(* CODESYS project CommonTypesAndFunctions 1.1.0.5.library
   Description: Some things to collect...
      some based on OSCAT library.
      see www.oscat.de for here home
   Version: 1.1.0.5
   Title: Common Helper for development
   Author: Stefan Dreyer
   DocFormat: reStructuredText
   Placeholder: CommonTypesAndFunctions
   LanguageModelAttribute: qualified-access-only
   CompiledLibraryCompatibilityVersion: CODESYS V3.5 SP15 Patch 2
   Company: Stefan Dreyer
   DefaultNamespace: CommonTypesAndFunctions

Project tree, tasks and I/O mapping:
  libraries: CAA Types Extern, * (CAA Technical Workgroup); CAA Behaviour Model, * (CAA Technical Workgroup); CAA FB Factory, * (CAA Technical Workgroup); SysTypes Interfaces, 3.5.2.0 (System); Time and Date, 3.5.7.0 (3S - Smart Software Solutions GmbH); SysTarget, 3.5.5.0 (System); SysMem, 3.5.12.0 (System); Standard, 3.5.15.0 (System); CmpErrors2 Interfaces, 3.5.15.0 (System); SysSem, 3.5.16.0 (System); SysProcess, 3.5.16.0 (System); Standard64, 3.5.16.0 (System); SysSocket2, 3.5.16.10 (System); CmpX509Cert, 3.5.15.0 (System); CmpTls, 3.5.15.0 (System); Base Interfaces, 3.5.2.0 (System); SysSocket, 3.5.15.0 (System); OSCAT Basic Extensions, 1.0.0.0 (Stefan Dreyer); BASIC, 3.3.4.0 (OSCAT); BUILDING, 1.0.0.1 (OSCAT); OSCAT Network Types, 1.0.0.1 (Stefan Dreyer)
  Common/
    Enums/
      data type ERROR
      data type VAR_TYPES
    Function Blocks/
      function block IP_CONTROL [ST]
      function block TIME_DATE_IMPULS [ST]
      function block TestString [ST]
      function block IP_CONTROL_TLS [ST]
      function block CounterToActuall [ST]: CounterInit, SetCounterResetImp
      function block StringImpact [ST]
      function block GetInstanceName [ST]: GetInstanceTopic, ReduceToLastNLevels, getLastName, GetName
      function block RELAIS_OUT_16_TRANSLATOR [ST]
      function block SmartDim [ST]
      function block Spratzel [ST]: setRand
      function block Rand [ST]: getRand
      Tests/
        function block TestNames1 [ST]
        function block TestInstanceName [ST]: FB_Init
        function block TestAnyX [ST]
      function block UpDown [ST]
      function block BLIND_INPUT_PERS [ST]
      function block BLIND_CONTROL_S_PERS [ST]
      function block BLIND_INPUT_EXT_PERS [ST]
      function block DivideByN [ST]
    Functions/
      function GET_DNS_IP [ST]
      function GetChar [ST]
      function find [ST]
      function len [ST]
      function concat [ST]
      function ResolveIPAddr [ST]
      function CheckDeltaValue [ST]
      function GetValueFromPointer [ST]
      function GetValueString [ST]
      function test [ST]
      function StrEquals [ST]
      function StrEqualsAtStart [ST]
      function GetValueFromStringPt [ST]
      function StrEqualsAtStartWithDelimiter [ST]
      function FindLastDot [ST]
      function MakeAllTypesPointer [ST]
      function GetJSONValue [ST]
      function Steps [ST]
      function GetValueStringFaktor [ST]
      function unionAdd [ST]
      function unionSub [ST]
      function unionMul [ST]
      function unionDiv [ST]
      function unionLimit [ST]
      function uint_to_Union [ST]
      function ScaleAllTypesUnion [ST]
      function AnyToUnion [ST]
      function unionToAny [ST]
      function checkJSON [ST]
    GlobalConstants/
      global variables MyConstants
    GlobalVariables/
      global variables Variables
    Interfaces/
    Structs/
      data type SMART_DIMM
      data type SMART_DIMM_ELEMENT
      data type IP_C_EXT
    Templates/
      Behaviour Model/
        function block ETrigA_Temp [ST]: prvAbort, prvCyclicAction, prvResetOutputs, prvStart
        function block ETrigTlA_Temp [ST]: prvAbort, prvCyclicAction, prvResetOutputs, prvStart
        function block ETrigTl_Temp [ST]: prvAbort, prvCyclicAction, prvResetOutputs, prvStart
        function block ETrigToA_Temp [ST]: prvAbort, prvCyclicAction, prvResetOutputs, prvStart
        function block ETrigToTlA_Temp [ST]: prvAbort, prvCyclicAction, prvResetOutputs, prvStart
        function block ETrigToTl_Temp [ST]: prvAbort, prvCyclicAction, prvResetOutputs, prvStart
        function block ETrigTo_Temp [ST]: prvAbort, prvCyclicAction, prvResetOutputs, prvStart
        function block ETrig_Temp [ST]: prvAbort, prvCyclicAction, prvResetOutputs, prvStart
        function block LTrig_Temp [ST]: prvAbort, prvCyclicAction, prvResetOutputs, prvStart
      FB Factory/
        function block CustomData [ST]
        function block CustomFB [ST]: prvInstInit
        function block CustomFBFactory_heap [ST]: Create, prvInstCount, prvInstPoolExtendsFactor, prvInstSize
        function block CustomFBFactory_static [ST]: Create, prvInstPoolAdr, prvInstPoolSize, prvInstSize
    Types/
      data type ALL_TYPES_UNION
      data type ALL_TYPES_UNION_POINTER
      data type EEPROM_DATA
      data type TIME_DATE_IMPULS_DATA
      data type TLS_CONFIG
      data type PWConfigs
      data type ENVIRONMENT_DATA
*)

// Common/Enums/ERROR
{attribute 'qualified_only'}
//{attribute 'conditionalshow'}
//{attribute 'conditionalshow' := 'SomeText'}
//{attribute 'hide'}
TYPE ERROR : (NO_ERROR, TIME_OUT); END_TYPE

// Common/Types/ALL_TYPES_UNION
TYPE ALL_TYPES_UNION :
UNION
	SINT_T:SINT;
	USINT_T:USINT;
	INT_T:INT;
	UINT_T:UINT;
	LINT_T:LINT;
	ULINT_T:ULINT;
	DINT_T:DINT;
	UDINT_T:UDINT;
	REAL_T:REAL;
	LREAL_T:LREAL;
	BYTE_T:BYTE;
	WORD_T:WORD;
	DWORD_T:DWORD;
	LWORD_T:LWORD;
	DT_T:DT;
	TIME_T:TIME;
	LTIME_T:LTIME;
	TOD_T:TOD;
	TOD_T2:ARRAY[0..1]OF TOD;
	DATE_T:DATE;
	BYTE_ARRAY:ARRAY[0..7]OF BYTE;
	BOOL_T:BOOL;
	
	//don't use strings UNION would be TO big....
END_UNION
END_TYPE

// Common/Types/ALL_TYPES_UNION_POINTER
TYPE ALL_TYPES_UNION_POINTER :
UNION
	POINTER_TO_SINT_T:POINTER TO SINT;
	POINTER_TO_USINT_T:POINTER TO USINT;
	POINTER_TO_INT_T:POINTER TO INT;
	POINTER_TO_UINT_T:POINTER TO UINT;
	POINTER_TO_LINT_T:POINTER TO LINT;
	POINTER_TO_ULINT_T:POINTER TO ULINT;
	POINTER_TO_DINT_T:POINTER TO DINT;
	POINTER_TO_UDINT_T:POINTER TO UDINT;
	POINTER_TO_REAL_T:POINTER TO REAL;
	POINTER_TO_LREAL_T:POINTER TO LREAL;
	POINTER_TO_BYTE_T:POINTER TO BYTE;
	POINTER_TO_WORD_T:POINTER TO WORD;
	POINTER_TO_DWORD_T:POINTER TO DWORD;
	POINTER_TO_LWORD_T:POINTER TO LWORD;
	POINTER_TO_DT_T:POINTER TO DT;
	POINTER_TO_TIME_T:POINTER TO TIME;
	POINTER_TO_LTIME_T:POINTER TO LTIME;
	POINTER_TO_TOD_T:POINTER TO TOD;
	POINTER_TO_TOD_T2:POINTER TO ARRAY[0..1]OF TOD;
	POINTER_TO_DATE_T:POINTER TO DATE;
	POINTER_TO_BYTE_ARRAY_T:POINTER TO ARRAY[0..7]OF BYTE;
	POINTER_TO_BOOL_T:POINTER TO BOOL;
	POINTER_TO_STRING_T: POINTER TO STRING(2000);

END_UNION
END_TYPE

// Common/Types/EEPROM_DATA
TYPE EEPROM_DATA :
STRUCT
	//FB_NO_AUTO:UINT;//auto createt FB NO, not possible because of multitasking ... so bad...
	FB_NO_IN:UINT;//allways check FB_IN_NO to be 0!!! so the EEPROM is free to do something!
	FB_NO_OUT:UINT;
	PAGE_IN:ARRAY[0..128-1] OF BYTE;
	PAGE_OUT:ARRAY[0..128-1] OF BYTE;
	READ_PAGE: BOOL;
	WRITE_PAGE: BOOL;
	ADDRESS_PAGE: UINT;
	ADDRESS_VALUE: UINT;
	VALUE_IN:ALL_TYPES_UNION;
	VALUE_OUT:ALL_TYPES_UNION; 
	READ_VALUE: BOOL;
	WRITE_VALUE: BOOL;
	PAGE_SIZE:UINT:=128;
	SIZE_OF_VALUE:UINT;
	SEMAPHORE:SysSem.RTS_IEC_HANDLE; //Semaphore for Consistence for EEPROM DATA is bus is out of main task
	HANDLE_VALID: BOOL;

END_STRUCT
END_TYPE

// Common/Types/TIME_DATE_IMPULS_DATA
TYPE TIME_DATE_IMPULS_DATA :
STRUCT
	
	IMP:BOOL;//1s impulse
	UDT:DT;//World Time
	SYSTEM_TIME:DT;//Time on SYSTEM
	TIME_IO:BOOL;//TIME IS I.O.
	TD_TIME:OSCAT_BASIC.SDT;
	//impulse at 00:00:00
	DAY_CHANGE:BOOL;
END_STRUCT
END_TYPE

// Common/Types/TLS_CONFIG
TYPE TLS_CONFIG :
STRUCT
	//see CmpTls for Doku of Method, initialisied to work as client
	tlsMethod: CmpTls.CmpTlsMethod := CmpTls.CmpTlsMethod.TLSv2_CLIENT;
	//List of allowed ciphers, initialised to medium, see openSSL for cipherList config
	chiperList:STRING(255) := 'HIGH';
	//certificates and ca still not supportet by CmpTls. So initialised to dont use certificats....
	{info 'here to implement certificate use'}
	verifyMode:DWORD := CmpTls.CmpTlsConstants.TLS_VERIFY_CLIENT_ONCE;
	
END_STRUCT
END_TYPE

// Common/Enums/VAR_TYPES
{attribute 'qualified_only'}
{attribute 'strict'}
TYPE VAR_TYPES :
(
	//enum_member := 0
	SINT_T, USINT_T, INT_T, UINT_T, DINT_T, UDINT_T, 
				LINT_T, ULINT_T, REAL_T, LREAL_T, BYTE_T, WORD_T,
				DWORD_T, LWORD_T, DT_T, TIME_T, TOD_T, TOD2_T, DATE_T, ARRAY_T, BOOL_T,
				STRING_T, LTIME_T
);
END_TYPE

// Common/Types/PWConfigs
TYPE PWConfigs :
STRUCT
PointerTo:ALL_TYPES_UNION_POINTER;
//PointerTo1:POINTER TO BYTE;
ValueType:VAR_TYPES;
NeedsMQTT:BOOL;
NeedsDB:BOOL;
MQTTTopic:POINTER TO STRING;
MQTTName:POINTER TO STRING;
MQTTDiff:UINT;
MQTTDezimal:INT;
MQTTTime:TIME;
MQTTRetain:BOOL;
MQTTQoS:SD_MQTT.QoS;
DBName:STRING;
DBNum:UINT;




END_STRUCT
END_TYPE

// Common/Structs/SMART_DIMM
TYPE SMART_DIMM :
STRUCT
	values:ARRAY[0..MyConstants.SMART_DIMM_STAGES-1] OF SMART_DIMM_ELEMENT;
END_STRUCT
END_TYPE

// Common/Structs/SMART_DIMM_ELEMENT
TYPE SMART_DIMM_ELEMENT :
STRUCT
	RunTime:TIME;//duration off effect
	DeltaOut:UINT;//Delta for Output
	_from:LREAL;
	_to:LREAL;
	Value:UINT;
END_STRUCT
END_TYPE

// Common/Types/ENVIRONMENT_DATA
TYPE ENVIRONMENT_DATA :
STRUCT
	//Possible Data from BME280 from Bosch Sensor Tec
	//using -->LREAL;
	Temperatur:LREAL;//using -->LREAL;
	//using -->LREAL;
	Humidity:LREAL;//using -->LREAL;
	//using -->LREAL;
	Pressure: LREAL;//using -->LREAL;
	//using -->REAL;
	absHumidity:REAL;//using -->REAL;
	//using -->REAL;
	dewPoint:REAL;//using -->REAL;


END_STRUCT
END_TYPE

// Common/Structs/IP_C_EXT
TYPE IP_C_EXT EXTENDS OSCAT_NETWORK_TYPES.IP_C :
STRUCT
	ResultSend:SysTypes.RTS_IEC_RESULT; 			(*Result of TCP Send call*)
	ResultReceive:SysTypes.RTS_IEC_RESULT;		(*Result of TCP Receive call*)
END_STRUCT
END_TYPE

// Common/GlobalConstants/MyConstants
{attribute 'qualified_only'}
//{attribute 'conditionalshow'}
//{attribute 'conditionalshow' := 'SomeText'}
//{attribute 'hide'}
VAR_GLOBAL CONSTANT
	gc_iDummy : INT := 42; /// This is a dummy global constant variable
	//Countrs in coutr ;)
	COUNTER_COUNT:UINT:=5;
	SMART_DIMM_STAGES:UINT:=5;
END_VAR

// Common/GlobalVariables/Variables
{attribute 'qualified_only'}
//{attribute 'conditionalshow'}
//{attribute 'conditionalshow' := 'SomeText'}
//{attribute 'hide'}
VAR_GLOBAL
	g_iDummy : INT; /// This is a dummy global variable
END_VAR

// Common/Templates/Behaviour Model/ETrigA_Temp
//{attribute 'hide_all_locals'}
//{attribute 'conditionalshow_all_locals' := 'SomeText'}
//{attribute 'conditionalshow_all_locals'}
//{attribute 'conditionalshow' := 'SomeText'}
//{attribute 'conditionalshow'}
//{attribute 'hide'}
FUNCTION_BLOCK ETrigA_Temp EXTENDS CBM.ETrigA
VAR_INPUT
	(* specific Inputs *)
END_VAR
VAR_OUTPUT
	eError : ERROR;
	(* specific Outputs *)
END_VAR
VAR
	(* specific vars *)
END_VAR

SUPER^();
IF iError = CBM.ERROR.TIME_OUT THEN
	eError := ERROR.TIME_OUT;
ELSE
	eError := iError;
END_IF

{attribute 'hide'}
METHOD prvAbort : BOOL
VAR_INPUT
END_VAR
VAR
END_VAR
IF xError THEN (* abort because of error *)
	(* TODO: insert specific Code here *)
ELSE (* user abort *)
	(* TODO: insert specific Code here *)
END_IF
xAbortInProgress:= FALSE;
END_METHOD

{attribute 'hide'}
METHOD prvCyclicAction : BOOL
VAR_INPUT
END_VAR
VAR
END_VAR
(* TODO: insert specific Code here *)
xDone:= TRUE;
(* if an error occurs, set iError to a value else than zero instead of xDone:= TRUE *)
(* to keep repeat loop *)
END_METHOD

{attribute 'hide'}
METHOD prvResetOutputs : BOOL
VAR_INPUT
END_VAR
VAR
END_VAR
(* TODO: insert specific Code here *)
SUPER^.prvResetOutputs();
END_METHOD

{attribute 'hide'}
METHOD prvStart : BOOL
VAR_INPUT
END_VAR
VAR
END_VAR
(* this code is called, when the application is started (rising edge of xExecute *)
(* TODO: copy specific input variables into local copies *)
(* TODO: insert specific Code here *)
;
END_METHOD

END_FUNCTION_BLOCK

// Common/Templates/Behaviour Model/ETrigTlA_Temp
//{attribute 'hide_all_locals'}
//{attribute 'conditionalshow_all_locals' := 'SomeText'}
//{attribute 'conditionalshow_all_locals'}
//{attribute 'conditionalshow' := 'SomeText'}
//{attribute 'conditionalshow'}
//{attribute 'hide'}
FUNCTION_BLOCK ETrigTlA_Temp EXTENDS CBM.ETrigTlA
VAR_INPUT
	(* specific Inputs *)
END_VAR
VAR_OUTPUT
	eError : ERROR;
	(* specific Outputs *)
END_VAR
VAR
	(* specific vars *)
END_VAR

SUPER^();
IF iError = CBM.ERROR.TIME_OUT THEN
	eError := ERROR.TIME_OUT;
ELSE
	eError := iError;
END_IF

{attribute 'hide'}
METHOD prvAbort : BOOL
VAR_INPUT
END_VAR
VAR
END_VAR
IF xError THEN (* abort because of error *)
	(* TODO: insert specific Code here *)
ELSE (* user abort *)
	(* TODO: insert specific Code here *)
END_IF
xAbortInProgress:= FALSE;
END_METHOD

{attribute 'hide'}
METHOD prvCyclicAction : BOOL
VAR_INPUT
END_VAR
VAR
END_VAR
(* TODO: insert specific Code here *)
xDone:= TRUE;
(* if an error occurs, set iError to a value else than zero instead of xDone:= TRUE *)
(* to keep repeat loop *)
END_METHOD

{attribute 'hide'}
METHOD prvResetOutputs : BOOL
VAR_INPUT
END_VAR
VAR
END_VAR
(* TODO: insert specific Code here *)
SUPER^.prvResetOutputs();
END_METHOD

{attribute 'hide'}
METHOD prvStart : BOOL
VAR_INPUT
END_VAR
VAR
END_VAR
(* this code is called, when the application is started (rising edge of xExecute *)
(* TODO: copy specific input variables into local copies *)
(* TODO: insert specific Code here *)
;
END_METHOD

END_FUNCTION_BLOCK

// Common/Templates/Behaviour Model/ETrigTl_Temp
//{attribute 'hide_all_locals'}
//{attribute 'conditionalshow_all_locals' := 'SomeText'}
//{attribute 'conditionalshow_all_locals'}
//{attribute 'conditionalshow' := 'SomeText'}
//{attribute 'conditionalshow'}
//{attribute 'hide'}
FUNCTION_BLOCK ETrigA_Temp EXTENDS CBM.ETrigTl
VAR_INPUT
	(* specific Inputs *)
END_VAR
VAR_OUTPUT
	eError : ERROR;
	(* specific Outputs *)
END_VAR
VAR
	(* specific vars *)
END_VAR

SUPER^();
IF iError = CBM.ERROR.TIME_OUT THEN
	eError := ERROR.TIME_OUT;
ELSE
	eError := iError;
END_IF

{attribute 'hide'}
METHOD prvAbort : BOOL
VAR_INPUT
END_VAR
VAR
END_VAR
IF xError THEN (* abort because of error *)
	(* TODO: insert specific Code here *)
ELSE (* user abort *)
	(* TODO: insert specific Code here *)
END_IF
xAbortInProgress:= FALSE;
END_METHOD

{attribute 'hide'}
METHOD prvCyclicAction : BOOL
VAR_INPUT
END_VAR
VAR
END_VAR
(* TODO: insert specific Code here *)
xDone:= TRUE;
(* if an error occurs, set iError to a value else than zero instead of xDone:= TRUE *)
(* to keep repeat loop *)
END_METHOD

{attribute 'hide'}
METHOD prvResetOutputs : BOOL
VAR_INPUT
END_VAR
VAR
END_VAR
(* TODO: insert specific Code here *)
SUPER^.prvResetOutputs();
END_METHOD

{attribute 'hide'}
METHOD prvStart : BOOL
VAR_INPUT
END_VAR
VAR
END_VAR
(* this code is called, when the application is started (rising edge of xExecute *)
(* TODO: copy specific input variables into local copies *)
(* TODO: insert specific Code here *)
;
END_METHOD

END_FUNCTION_BLOCK

// Common/Templates/Behaviour Model/ETrigToA_Temp
//{attribute 'hide_all_locals'}
//{attribute 'conditionalshow_all_locals' := 'SomeText'}
//{attribute 'conditionalshow_all_locals'}
//{attribute 'conditionalshow' := 'SomeText'}
//{attribute 'conditionalshow'}
//{attribute 'hide'}
FUNCTION_BLOCK ETrigToA_Temp EXTENDS CBM.ETrigToA
VAR_INPUT
	(* specific Inputs *)
END_VAR
VAR_OUTPUT
	eError : ERROR;
	(* specific Outputs *)
END_VAR
VAR
	(* specific vars *)
END_VAR

SUPER^();
IF iError = CBM.ERROR.TIME_OUT THEN
	eError := ERROR.TIME_OUT;
ELSE
	eError := iError;
END_IF

{attribute 'hide'}
METHOD prvAbort : BOOL
VAR_INPUT
END_VAR
VAR
END_VAR
IF xError THEN (* abort because of error *)
	(* TODO: insert specific Code here *)
ELSE (* user abort *)
	(* TODO: insert specific Code here *)
END_IF
xAbortInProgress:= FALSE;
END_METHOD

{attribute 'hide'}
METHOD prvCyclicAction : BOOL
VAR_INPUT
END_VAR
VAR
END_VAR
(* TODO: insert specific Code here *)
xDone:= TRUE;
(* if an error occurs, set iError to a value else than zero instead of xDone:= TRUE *)
END_METHOD

{attribute 'hide'}
METHOD prvResetOutputs : BOOL
VAR_INPUT
END_VAR
VAR
END_VAR
(* TODO: insert specific Code here *)
SUPER^.prvResetOutputs();
END_METHOD

{attribute 'hide'}
METHOD prvStart : BOOL
VAR_INPUT
END_VAR
VAR
END_VAR
(* this code is called, when the application is started (rising edge of xExecute *)
(* TODO: copy specific input variables into local copies *)
(* TODO: insert specific Code here *)
;
END_METHOD

END_FUNCTION_BLOCK

// Common/Templates/Behaviour Model/ETrigToTlA_Temp
//{attribute 'hide_all_locals'}
//{attribute 'conditionalshow_all_locals' := 'SomeText'}
//{attribute 'conditionalshow_all_locals'}
//{attribute 'conditionalshow' := 'SomeText'}
//{attribute 'conditionalshow'}
//{attribute 'hide'}
FUNCTION_BLOCK ETrigToTlA_Temp EXTENDS CBM.ETrigToTlA
VAR_INPUT
	(* specific Inputs *)
END_VAR
VAR_OUTPUT
	eError : ERROR;
	(* specific Outputs *)
END_VAR
VAR
	(* specific vars *)
END_VAR

SUPER^();
IF iError = CBM.ERROR.TIME_OUT THEN
	eError := ERROR.TIME_OUT;
ELSE
	eError := iError;
END_IF

{attribute 'hide'}
METHOD prvAbort : BOOL
VAR_INPUT
END_VAR
VAR
END_VAR
IF xError THEN (* abort because of error *)
	(* TODO: insert specific Code here *)
ELSE (* user abort *)
	(* TODO: insert specific Code here *)
END_IF
xAbortInProgress:= FALSE;
END_METHOD

{attribute 'hide'}
METHOD prvCyclicAction : BOOL
VAR_INPUT
END_VAR
VAR
END_VAR
(* TODO: insert specific Code here *)
xDone:= TRUE;
(* if an error occurs, set iError to a value else than zero instead of xDone:= TRUE *)
(* to keep repeat loop *)
END_METHOD

{attribute 'hide'}
METHOD prvResetOutputs : BOOL
VAR_INPUT
END_VAR
VAR
END_VAR
(* TODO: insert specific Code here *)
SUPER^.prvResetOutputs();
END_METHOD

{attribute 'hide'}
METHOD prvStart : BOOL
VAR_INPUT
END_VAR
VAR
END_VAR
(* this code is called, when the application is started (rising edge of xExecute *)
(* TODO: copy specific input variables into local copies *)
(* TODO: insert specific Code here *)
;
END_METHOD

END_FUNCTION_BLOCK

// Common/Templates/Behaviour Model/ETrigToTl_Temp
//{attribute 'hide_all_locals'}
//{attribute 'conditionalshow_all_locals' := 'SomeText'}
//{attribute 'conditionalshow_all_locals'}
//{attribute 'conditionalshow' := 'SomeText'}
//{attribute 'conditionalshow'}
//{attribute 'hide'}
FUNCTION_BLOCK ETrigToTl_Temp EXTENDS CBM.ETrigToTl
VAR_INPUT
	(* specific Inputs *)
END_VAR
VAR_OUTPUT
	eError : ERROR;
	(* specific Outputs *)
END_VAR
VAR
	(* specific vars *)
END_VAR

SUPER^();
IF iError = CBM.ERROR.TIME_OUT THEN
	eError := ERROR.TIME_OUT;
ELSE
	eError := iError;
END_IF

{attribute 'hide'}
METHOD prvAbort : BOOL
VAR_INPUT
END_VAR
VAR
END_VAR
IF xError THEN (* abort because of error *)
	(* TODO: insert specific Code here *)
ELSE (* user abort *)
	(* TODO: insert specific Code here *)
END_IF
xAbortInProgress:= FALSE;
END_METHOD

{attribute 'hide'}
METHOD prvCyclicAction : BOOL
VAR_INPUT
END_VAR
VAR
END_VAR
(* TODO: insert specific Code here *)
xDone:= TRUE;
(* if an error occurs, set iError to a value else than zero instead of xDone:= TRUE *)
(* to keep repeat loop *)
END_METHOD

{attribute 'hide'}
METHOD prvResetOutputs : BOOL
VAR_INPUT
END_VAR
VAR
END_VAR
(* TODO: insert specific Code here *)
SUPER^.prvResetOutputs();
END_METHOD

{attribute 'hide'}
METHOD prvStart : BOOL
VAR_INPUT
END_VAR
VAR
END_VAR
(* this code is called, when the application is started (rising edge of xExecute *)
(* TODO: copy specific input variables into local copies *)
(* TODO: insert specific Code here *)
;
END_METHOD

END_FUNCTION_BLOCK

// Common/Templates/Behaviour Model/ETrigTo_Temp
//{attribute 'hide_all_locals'}
//{attribute 'conditionalshow_all_locals' := 'SomeText'}
//{attribute 'conditionalshow_all_locals'}
//{attribute 'conditionalshow' := 'SomeText'}
//{attribute 'conditionalshow'}
//{attribute 'hide'}
FUNCTION_BLOCK ETrigTo_Temp EXTENDS CBM.ETrigTo
VAR_INPUT
	(* specific Inputs *)
END_VAR
VAR_OUTPUT
	eError : ERROR;
	(* specific Outputs *)
END_VAR
VAR
	(* specific vars *)
END_VAR

SUPER^();
IF iError = CBM.ERROR.TIME_OUT THEN
	eError := ERROR.TIME_OUT;
ELSE
	eError := iError;
END_IF

{attribute 'hide'}
METHOD prvAbort : BOOL
VAR_INPUT
END_VAR
VAR
END_VAR
IF xError THEN (* abort because of error *)
	(* TODO: insert specific Code here *)
ELSE (* user abort *)
	(* TODO: insert specific Code here *)
END_IF
xAbortInProgress:= FALSE;
END_METHOD

{attribute 'hide'}
METHOD prvCyclicAction : BOOL
VAR_INPUT
END_VAR
VAR
END_VAR
(* TODO: insert specific Code here *)
xDone:= TRUE;
(* if an error occurs, set iError to a value else than zero instead of xDone:= TRUE *)
(* to keep repeat loop *)
END_METHOD

{attribute 'hide'}
METHOD prvResetOutputs : BOOL
VAR_INPUT
END_VAR
VAR
END_VAR
(* TODO: insert specific Code here *)
SUPER^.prvResetOutputs();
END_METHOD

{attribute 'hide'}
METHOD prvStart : BOOL
VAR_INPUT
END_VAR
VAR
END_VAR
(* this code is called, when the application is started (rising edge of xExecute *)
(* TODO: copy specific input variables into local copies *)
(* TODO: insert specific Code here *)
;
END_METHOD

END_FUNCTION_BLOCK

// Common/Templates/Behaviour Model/ETrig_Temp
//{attribute 'hide_all_locals'}
//{attribute 'conditionalshow_all_locals' := 'SomeText'}
//{attribute 'conditionalshow_all_locals'}
//{attribute 'conditionalshow' := 'SomeText'}
//{attribute 'conditionalshow'}
//{attribute 'hide'}
FUNCTION_BLOCK ETrig_Temp EXTENDS CBM.ETrig
VAR_INPUT
	(* specific Inputs *)
END_VAR
VAR_OUTPUT
	eError : ERROR;
	(* specific Outputs *)
END_VAR
VAR
	(* specific vars *)
END_VAR

SUPER^();
IF iError = CBM.ERROR.TIME_OUT THEN
	eError := ERROR.TIME_OUT;
ELSE
	eError := iError;
END_IF

{attribute 'hide'}
METHOD prvAbort : BOOL
VAR_INPUT
END_VAR
VAR
END_VAR
IF xError THEN (* abort because of error *)
	(* TODO: insert specific Code here *)
ELSE (* user abort *)
	(* TODO: insert specific Code here *)
END_IF
xAbortInProgress:= FALSE;
END_METHOD

{attribute 'hide'}
METHOD prvCyclicAction : BOOL
VAR_INPUT
END_VAR
VAR
END_VAR
(* TODO: insert specific Code here *)
xDone:= TRUE;
(* if an error occurs, set iError to a value else than zero instead of xDone:= TRUE *)
(* to keep repeat loop *)
END_METHOD

{attribute 'hide'}
METHOD prvResetOutputs : BOOL
VAR_INPUT
END_VAR
VAR
END_VAR
(* TODO: insert specific Code here *)
SUPER^.prvResetOutputs();
END_METHOD

{attribute 'hide'}
METHOD prvStart : BOOL
VAR_INPUT
END_VAR
VAR
END_VAR
(* this code is called, when the application is started (rising edge of xExecute *)
(* TODO: copy specific input variables into local copies *)
(* TODO: insert specific Code here *)
;
END_METHOD

END_FUNCTION_BLOCK

// Common/Templates/Behaviour Model/LTrig_Temp
//{attribute 'hide_all_locals'}
//{attribute 'conditionalshow_all_locals' := 'SomeText'}
//{attribute 'conditionalshow_all_locals'}
//{attribute 'conditionalshow' := 'SomeText'}
//{attribute 'conditionalshow'}
//{attribute 'hide'}
FUNCTION_BLOCK LTrig_Temp EXTENDS CBM.LTrig
VAR_INPUT
	(* specific Inputs *)
END_VAR
VAR_OUTPUT
	eError : ERROR;
	(* specific Outputs *)
END_VAR
VAR
	(* specific vars *)
END_VAR

SUPER^();
IF iError = CBM.ERROR.TIME_OUT THEN
	eError := ERROR.TIME_OUT;
ELSE
	eError := iError;
END_IF

{attribute 'hide'}
METHOD prvAbort : BOOL
VAR_INPUT
END_VAR
VAR
END_VAR
IF xError THEN (* abort because of error *)
	(* TODO: insert specific Code here *)
ELSE (* user abort *)
	(* TODO: insert specific Code here *)
END_IF
xAbortInProgress:= FALSE;
END_METHOD

{attribute 'hide'}
METHOD prvCyclicAction : BOOL
VAR_INPUT
END_VAR
VAR
END_VAR
(* TODO: insert specific Code here *)
xDone:= TRUE;
(* if an error occurs, set iError to a value else than zero instead of xDone:= TRUE *)
(* to keep repeat loop *)
END_METHOD

{attribute 'hide'}
METHOD prvResetOutputs : BOOL
VAR_INPUT
END_VAR
VAR
END_VAR
(* TODO: insert specific Code here *)
SUPER^.prvResetOutputs();
END_METHOD

{attribute 'hide'}
METHOD prvStart : BOOL
VAR_INPUT
END_VAR
VAR
END_VAR
(* this code is called, when the application is started (rising edge of xExecute *)
(* TODO: copy specific input variables into local copies *)
(* TODO: insert specific Code here *)
;
END_METHOD

END_FUNCTION_BLOCK

// Common/Templates/FB Factory/CustomData
// This is a container to carry init data from the Create methode of the factory
// to the prvInstInit methode of the new generated function block instance
{attribute 'enable_dynamic_creation'}
//{attribute 'hide_all_locals'}
//{attribute 'conditionalshow_all_locals' := 'SomeText'}
//{attribute 'conditionalshow_all_locals'}
//{attribute 'conditionalshow' := 'SomeText'}
//{attribute 'conditionalshow'}
//{attribute 'hide'}
FUNCTION_BLOCK CustomData EXTENDS FBF.InstanceData
VAR_INPUT
	(* Todo: Add your application specific data as input variables *)
END_VAR

(* !! Do not add any executable code here !! *)
SUPER^();

END_FUNCTION_BLOCK

// Common/Templates/FB Factory/CustomFB
{attribute 'enable_dynamic_creation'}
//{attribute 'hide_all_locals'}
//{attribute 'conditionalshow_all_locals' := 'SomeText'}
//{attribute 'conditionalshow_all_locals'}
//{attribute 'conditionalshow' := 'SomeText'}
//{attribute 'conditionalshow'}
//{attribute 'hide'}
FUNCTION_BLOCK CustomFB EXTENDS FBF.InstanceBase;
VAR_INPUT
END_VAR
VAR_OUTPUT
END_VAR
VAR
END_VAR

SUPER^();

// This methode is called from the factory to give a chance
// to initialize the new fb instance with the content of itfData
//{attribute 'hide_all_locals'}
//{attribute 'conditionalshow_all_locals' := 'SomeText'}
//{attribute 'conditionalshow_all_locals'}
//{attribute 'conditionalshow' := 'SomeText'}
//{attribute 'conditionalshow'}
//{attribute 'hide'}
METHOD prvInstInit : FBF.ERROR
VAR_INPUT
	itfData : FBF.IData; 
END_VAR
VAR
	pData : POINTER TO CustomData;
	xOk : BOOL;
END_VAR
SUPER^.prvInstInit(itfData);
xOk := __QUERYPOINTER(itfData, pData);
IF xOk THEN
	(* THIS^.iLocalVar := pData^.iInitValue *);
END_IF
END_METHOD

END_FUNCTION_BLOCK

// Common/Templates/FB Factory/CustomFBFactory_heap
// This is a template for a factory with an heap based extendable memory pool
{attribute 'enable_dynamic_creation'}
//{attribute 'hide_all_locals'}
//{attribute 'conditionalshow_all_locals' := 'SomeText'}
//{attribute 'conditionalshow_all_locals'}
//{attribute 'conditionalshow' := 'SomeText'}
//{attribute 'conditionalshow'}
//{attribute 'hide'}
FUNCTION_BLOCK CustomFBFactory_heap EXTENDS FBF.FactoryBase
VAR
END_VAR

SUPER^();

(* Please replace CustonFB with your specific function block type *)
(* There is no need to change anything else !!! *)
METHOD Create : POINTER TO CustomFB
VAR_INPUT
	itfData : FBF.IData;
END_VAR
VAR_OUTPUT
	eError : FBF.ERROR;
END_VAR
VAR
	hInst : CAA.HANDLE;
	itfInst : FBF.IInstance;
	xOk : BOOL;
END_VAR
(* !!! This code must not be subject to change !!! *)
hInst := SUPER^.prvAllocInstMem(eError => eError);
Create := SUPER^.prvGetInstPointer(hInst);
IF Create <> 0 AND eError = FBF.ERROR.NO_ERROR THEN

	{implicit on}
	Create^.__vfInit();
	Create^.FB_Init(TRUE, FALSE);
	{implicit off}

	xOk := __QUERYINTERFACE(Create^, itfInst);
	IF xOk THEN
		xOk := SUPER^.prvInstInit(itfInst, hInst, itfData, eError=>eError);
	ELSE
		eError := FBF.ERROR.WRONG_INTERFACE;
	END_IF

	IF NOT xOk THEN
		SUPER^.prvFreeInstMem(hInst);
		Create := CAA.gc_pNULL;
	END_IF
END_IF
END_METHOD

//{attribute 'conditionalshow' := 'SomeText'}
//{attribute 'conditionalshow'}
//{attribute 'hide'}
PROPERTY prvInstCount : CAA.COUNT (* ctInst *)
GET
(* Please choose a proper value for prvInstCount *)
prvInstCount := 10;
END_GET
END_PROPERTY

//{attribute 'conditionalshow' := 'SomeText'}
//{attribute 'conditionalshow'}
//{attribute 'hide'}
PROPERTY prvInstPoolExtendsFactor : USINT (* usiFactor [0..x%] *)
GET
(* Please choose a proper value for prvInstPoolExtendsFactor *)
(* This value will be interpreted as a 0..x% size extendsion related to the original size of the pool *)
prvInstPoolExtendsFactor := 20;
END_GET
END_PROPERTY

//{attribute 'conditionalshow' := 'SomeText'}
//{attribute 'conditionalshow'}
//{attribute 'hide'}
PROPERTY prvInstSize : CAA.SIZE (* szInst *)
GET
(* Please replace CustomFB with your specific function block type *)
prvInstSize := sizeof(CustomFB);
END_GET
END_PROPERTY

END_FUNCTION_BLOCK

// Common/Templates/FB Factory/CustomFBFactory_static
// This is a template for a factory with an static iec memory based memory pool which a fixed capacity
{attribute 'enable_dynamic_creation'}
//{attribute 'hide_all_locals'}
//{attribute 'conditionalshow_all_locals' := 'SomeText'}
//{attribute 'conditionalshow_all_locals'}
//{attribute 'conditionalshow' := 'SomeText'}
//{attribute 'conditionalshow'}
//{attribute 'hide'}
FUNCTION_BLOCK CustomFBFactory_static EXTENDS FBF.FactoryBase
VAR
	// Please change the size of abyPoolMemory with your specific application need
	abyPoolMemory : ARRAY[0..529] OF BYTE;
END_VAR

SUPER^();

(* Please replace CustonFB with our specific function block type *)
(* There is no need to change anything else !!! *)
METHOD Create : POINTER TO CustomFB
VAR_INPUT
	itfData : FBF.IData;
END_VAR
VAR_OUTPUT
	eError : FBF.ERROR;
END_VAR
VAR
	hInst : CAA.HANDLE;
	itfInst : FBF.IInstance;
	xOk : BOOL;
END_VAR
(* !!! This code must not be subject to change !!! *)
hInst := SUPER^.prvAllocInstMem(eError => eError);
Create := SUPER^.prvGetInstPointer(hInst);
IF Create <> 0 AND eError = FBF.ERROR.NO_ERROR THEN

	{implicit on}
	Create^.__vfInit();
	Create^.FB_Init(TRUE, FALSE);
	{implicit off}

	xOk := __QUERYINTERFACE(Create^, itfInst);
	IF xOk THEN
		xOk := SUPER^.prvInstInit(itfInst, hInst, itfData, eError=>eError);
	ELSE
		eError := FBF.ERROR.WRONG_INTERFACE;
	END_IF

	IF NOT xOk THEN
		SUPER^.prvFreeInstMem(hInst);
		Create := CAA.gc_pNULL;
	END_IF
END_IF
END_METHOD

//{attribute 'conditionalshow' := 'SomeText'}
//{attribute 'conditionalshow'}
//{attribute 'hide'}
PROPERTY prvInstPoolAdr : CAA.PVOID (* pPool *)
GET
prvInstPoolAdr := ADR(abyPoolMemory);
END_GET
END_PROPERTY

//{attribute 'conditionalshow' := 'SomeText'}
//{attribute 'conditionalshow'}
//{attribute 'hide'}
PROPERTY prvInstPoolSize : CAA.SIZE (* szPool *)
GET
prvInstPoolSize := sizeof(abyPoolMemory);
END_GET
END_PROPERTY

//{attribute 'conditionalshow' := 'SomeText'}
//{attribute 'conditionalshow'}
//{attribute 'hide'}
PROPERTY prvInstSize : CAA.SIZE (* szInst *)
GET
(* Please replace CustomFB with your specific function block type *)
prvInstSize := sizeof(CustomFB);
END_GET
END_PROPERTY

END_FUNCTION_BLOCK

// Common/Function Blocks/IP_CONTROL
FUNCTION_BLOCK IP_CONTROL
VAR_IN_OUT
	IP_C : IP_C_EXT; (* IP_Control Verwaltungsstruktur *)
	S_BUF : OSCAT_NETWORK_TYPES.NETWORK_BUFFER; (* Externer Sendbuffer *)
	R_BUF : OSCAT_NETWORK_TYPES.NETWORK_BUFFER; (* Externer Receivebuffer *)
END_VAR
VAR_INPUT
	IP : DWORD; (* IP Adresse *)
	PORT : WORD; (* Port Nummer *)
	TIME_OUT : TIME; (* Ueberwachungszeit Connect / Send / Receive *)

END_VAR
VAR
	TLS_CONFIG:POINTER TO TLS_CONFIG;
	c_time : UDINT; (* CONNECT-Time (Zeit bei nicht vorhandener Verbindung) *)
	s_time : UDINT; (* SEND-Time    (Zeit seit letzten Datensenden) *)
	r_time : UDINT; (* RECEIVE-Time (Zeit seit letztem Datenempfang) *)

	c_enable : BOOL; (* Connect: freigabe *)
	c_ip : DWORD; (* Connect: aktuelle IP-Adresse *)
	c_port : WORD; (* Connect: aktuelle Port-Nummer *)
	c_mode : BYTE; (* Connect: aktueller Mode UDP/TCP...... *)
	c_status : BYTE; (* Connect: Status (Errorcode) *)
	c_ready : BOOL; (* Connect: Verbindung aufgebaut *)
	c_ready_old : BOOL; (* Connect: letzter Zustand von c_ready für Flankenauswertung *)
	c_select : BOOL; (* non blocking mode - abfrage über select durchführen *)
	c_fdWrite :  SysSocket2.SOCKET_FD_SET;
	c_Timeout : SysSocket2.SOCKET_TIMEVAL;
	//use a TLS connection
	TLS: BOOL;

		
	s_total : INT; (* Send: Gesamtanzahl Bytes zum senden *)
	s_cur_pos : INT; (* Send: aktuelle Sendeposition *)
	s_cur_size : INT; (* Send: aktuelle Sendegroesse *)
	s_max_size : INT; (* Send: maximale Telegrammlänge fuer Senden *)
	s_start : BOOL; (* Send: Sende modus aktivieren *)
	s_active : BOOL; (* Send: Daten senden ist aktiv *)
	s_req : BOOL; (* Send: Start Daten senden *)
	s_done : BOOL; (* Send: ohne Fehler beendet *)
	s_status : BYTE; (* Send: Status (Errorcodes) *)

	r_status : BYTE; (* Receive: Status (Errorcodes) *)
	r_count : INT; (* Receive: Anzahl empfangener Bytes *)
	r_offset : INT; (* Receive: aktuelle Position in externen Receivebuffer *)
	r_max_size : INT; (* Receive: groesse des externen Empfangbuffers*)

	new_connection : BOOL; (* Neue Verbindungsparameter vorhanden *)
	tx : DWORD; (* letzter zeitwert *)
	error_time : DWORD; (* aktueller Timeout-Wert *)
	//Socket Parameter
	SysSockParameter:SysSocket2.SysSocket2_Parameter;
	SysSockSpec : SysSocket2.SysSocket2_SpecificParameter;
	state: BYTE; (* schrittmerker für connect *)
	server_socket : SysTypes.RTS_IEC_HANDLE:= SysTypes.RTS_INVALID_HANDLE;                // Handle Pointing to our Socket
	socket : SysTypes.RTS_IEC_HANDLE:= SysTypes.RTS_INVALID_HANDLE;
	//TlsHandle := RTS_IEC_HANDLE:= RTS_INVALID_HANDLE;
	//server_socket : DINT:= RTS_INVALID_HANDLE;
	//socket : DINT:= RTS_INVALID_HANDLE;
	sockaddr : SysSocket2.SOCKADDRESS;
	sockaddrUDP : SysSocket.SOCKADDRESS;
	sockaddr_size : DWORD;
	plc_841 : BOOL;
	plc_881 : BOOL;
	dint_true : DINT := 1;
	dint_false : DINT := 0;
	bytes_received : DINT;
	bytes_sent : DINT;
	udp_mode : BOOL;

	pResult : SysTypes.RTS_IEC_RESULT; //Needed for V3 Lib
	FunctionResult 	: UDINT ;
	//tAddress                	: INADDR;                           // Strucutre to define our internet address
	//TESTtAddress               	: INADDR;   
	(*LOG_MSG : LOG_MSG;
	_debug_enable : BOOL := TRUE;
	debug_index : INT;
	debug_ID : INT;
	debug_lasterror : DWORD;
	debug_last_id : INT := 255;
	state_last: BYTE;*)
	
	TlsConnectTime:DWORD;
	TlsConnectLastTick:DWORD;
		
END_VAR

VAR CONSTANT
	STOP : BYTE := 0;
	TS_INIT: BYTE := 1;
	TS_OPEN : BYTE:= 2;

	UDP_INIT : BYTE:= 31;

	TC_INIT : BYTE:= 51;
	TC_CONNECT : BYTE:= 52;

	C_WAIT : BYTE:= 250;
	C_CLOSE : BYTE:= 251;
	

END_VAR

(*

version 1.9		26. Feb. 2012
programmer 		ks
tested by			ks

IP_CONTROL ist ein Wrapper-Baustein um eine Hersteller neutrale Schnittstelle zum Ethernet zu schaffen
*)

(* ---------------------- Debug-Message ----------------------------*)
(*IF _debug_enable THEN
	IF IP_C.FIFO.ID > BYTE#0 THEN (* nur wenn Teilnehmer ID's vorhanden sind *)
		debug_index := IP_C.FIFO.NR;
		debug_ID := BYTE_TO_INT(IP_C.FIFO.X[debug_index]);
	END_IF;
END_IF;*)
(* -----------------------------------------------------------------------------*)

(* read system time *)
tx := OSCAT_BASIC.T_PLC_MS();

IF IP_C.C_PORT = 0 THEN
	IP_C.C_PORT := PORT; (* uebergebenen PORT durch parametrierten PORT ersetzen *)
END_IF;
IF IP_C.C_IP = 0 AND IP_C.C_MODE < 4 THEN
	IP_C.C_IP := IP; (* uebergebene IP durch paramtrierte IP ersetzen *)
END_IF;

new_connection := c_ip <> IP_C.C_IP OR c_mode <> (IP_C.C_MODE AND 2#1111111) OR c_port <> IP_C.C_PORT; (* neue Verbindungs erwünscht ? *)
c_enable := IP_C.C_ENABLE AND NOT new_connection;

IF IP_C.C_ENABLE AND IP_C.ERROR = 0 AND state = STOP THEN (* Freigabe,kein Fehler,kein Socket offen *)
	c_ip   := IP_C.C_IP;
	c_mode := IP_C.C_MODE AND 2#1111111; //bit 7 for TLS Mode
	//TLS := IP_C.C_MODE.7;
	c_port := IP_C.C_PORT;
	plc_841 := ADR(%MW0)=16#30000000; (*750-841*)
	plc_881 := ADR(%MW0)=16#20000000; (*750-881*)
	udp_mode := C_MODE.0; (* Mode 1,3,5 = udp *)

	error_time := TIME_TO_DWORD(MAX(T#200ms,TIME_OUT));
	IP_C.TIME_RESET := TRUE; (* Alle Timer ruecksetzen *)

	r_max_size := UINT_TO_INT(SIZEOF(R_BUF.BUFFER));
	s_max_size := UINT_TO_INT(SIZEOF(S_BUF.BUFFER));

	IF C_MODE.0 THEN (* Mode: 1,3,5 = UDP CLIENT/SERVER *)
		state := UDP_INIT;
	ELSIF C_MODE = 0 THEN (* Mode: 0 = TCP CLIENT *)
		state := TC_INIT;
	ELSE
		state := TS_INIT; (* Mode: 2,4 = TCP SERVER *)
	END_IF;

	(* ---------------------- Debug-Message ----------------------------*)
	(*IF _debug_enable THEN
		LOG_CL.NEW_MSG := 'IP_CON: MODE ~1 / IP ~2 / PORT ~3 /ID ~6';
		LOG_CL.PRINTF[1] := BYTE_TO_STRING(C_MODE);
		LOG_CL.PRINTF[2] := IP4_TO_STRING(c_ip);
		LOG_CL.PRINTF[3] := WORD_TO_STRING(c_port);
		LOG_CL.PRINTF[6] := INT_TO_STRING(debug_ID);
		LOG_MSG();
	END_IF;*)
	(* -----------------------------------------------------------------------------*)

END_IF;

(* ---------------------- Debug-Message ----------------------------*)
(*IF  _debug_enable THEN
	IF state <> state_last THEN
		LOG_CL.NEW_MSG := 'IP_STEP ~1 -IP_ID ~6';
		LOG_CL.PRINTF[1] := BYTE_TO_STRING(state);
		LOG_CL.PRINTF[6] := INT_TO_STRING(debug_ID);
		LOG_MSG();
		state_last := state;
	END_IF;
END_IF;*)
(* -----------------------------------------------------------------------------*)

IF IP_C.TIME_RESET THEN (* Alle Timer ruecksetzen *)
	IP_C.TIME_RESET := FALSE; (* Reset rücksetzen *)
	c_time := tx; (* Connect Timer ruecksetzen *)
	s_time := tx; (* Send Timer ruecksetzen *)
	r_time := tx; (* Receive Timer ruecksetzen *)

	c_status := BYTE#0; (* letzten Connect Fehler rücksetzen *)
	s_status := BYTE#0; (* letzten Send Fehler rücksetzen *)
	r_status := BYTE#0; (* letzten Receive Fehler rücksetzen *)
END_IF;

(* ---------------------------------------------- *)

CASE state OF

UDP_INIT: (* UDP_CLIENT + SERVER *)
	//socket := SysSock2Create(SOCKET_AF_INET, SOCKET_DGRAM, SOCKET_IPPROTO_IP, ADR(pResult));
	(*SysSockParameter.parameterType := SysSocket2.SysSocket2_Type.STD;
	SysSockSpec.stdSockets.i32AddressFamily := SOCKET_AF_INET;
	SysSockSpec.stdSockets.i32Type := SOCKET_DGRAM;
	SysSockSpec.stdSockets.i32Protocol := SOCKET_IPPROTO_IP;
	SysSockParameter.specific := SysSockSpec;
	socket := SysSocket2.SysSock2Create(pParameter:= ADR(SysSockParameter), pResult:= ADR(pResult));*)	
	socket := SysSocket.SysSockCreate(SysSocket.GVL.SOCKET_AF_INET, SysSocket.GVL.SOCKET_DGRAM, SysSocket.GVL.SOCKET_IPPROTO_IP, ADR(pResult));
	IF socket < 0 THEN
		c_status := 1; (* SysSock2Create failed *)
		state := C_CLOSE;
	ELSE
		FunctionResult :=SysSocket.SysSockSetOption(socket, SysSocket.GVL.SOCKET_SOL, SysSocket.GVL.SOCKET_SO_BROADCAST, ADR(dint_true), SIZEOF(dint_true)); (* allow broadcast *)
		FunctionResult :=SysSocket.SysSockIoctl(socket, SysSocket.GVL.SOCKET_FIONBIO, ADR(dint_true)); (* put socket in non-blocking mode *)
		sockaddrUDP.sin_family := SysSocket.GVL.SOCKET_AF_INET;
		sockaddrUDP.sin_port := SysSocket.SysSockHtons(c_port);
		sockaddrUDP.sin_addr.ulAddr := SEL(c_mode = 1, SysSocket.GVL.SOCKET_INADDR_ANY, SysSocket.SysSockNtohl(c_ip));

		IF c_mode >= 2 THEN (* SERVER Mode *)
			FunctionResult := SysSocket.SysSockBind(socket, ADR(sockaddrUDP), SIZEOF(sockaddrUDP));
			IF FunctionResult=0 THEN
				c_ready := TRUE; (* Connected *)
				state:= C_WAIT;
			ELSE
				c_status := 2; (* SysSock2Bind failed *)
				state := C_CLOSE;
			END_IF;
		ELSE
			c_ready := TRUE; (* Connected *)
			state:= C_WAIT;
		END_IF;
	END_IF;
	

(* ---------------------------------------------- *)

TC_INIT: (* TCP-CLIENT (AKTIV) *)
	// Create handle to ethernet socket to send messages
	//socket        := SysSock2Create(SOCKET_AF_INET, SOCKET_STREAM, SOCKET_IPPROTO_TCP, ADR(pResult)); 
	IF TLS THEN
		SysSockParameter.parameterType := SysSocket2.SysSocket2_Type.TLS;
		SysSockSpec.tlsSockets.hTlsContext := CmpTls.CmpTlsCreateContext(
			hCert:= SysTypes.RTS_INVALID_HANDLE, 
			tlsMethod:= TLS_CONFIG^.tlsMethod, 
			cipherList:= ADR(TLS_CONFIG^.chiperList),
			verifyMode := TLS_CONFIG^.verifyMode,
			pResult:= ADR(pResult));
			SysSockParameter.specific := SysSockSpec;	
	ELSE
		SysSockParameter.parameterType := SysSocket2.SysSocket2_Type.STD;
		SysSockSpec.stdSockets.i32AddressFamily := SysSocket2.GVL.SOCKET_AF_INET;
		SysSockSpec.stdSockets.i32Type := SysSocket2.GVL.SOCKET_STREAM;
		SysSockSpec.stdSockets.i32Protocol := SysSocket2.GVL.SOCKET_IPPROTO_TCP;
		SysSockParameter.specific := SysSockSpec;	
	END_IF
	
	
	socket := SysSocket2.SysSock2Create(pParameter:= ADR(SysSockParameter), pResult:= ADR(pResult));	
	IF socket < 0 OR pResult <> CmpErrors.Errors.ERR_OK THEN
		c_status := 1;  (* SysSock2Create failed *)
		state := C_CLOSE;
	ELSE
		IF plc_841 OR plc_881 THEN
			FunctionResult := SysSocket2.SysSock2SetOption(socket,6,SysSocket2.GVL.SOCKET_TCP_NODELAY, ADR(dint_true), SIZEOF(dint_true)); (* Set Push-Bit *)
		END_IF;
		// Set option for local address reuse
		FunctionResult := SysSocket2.SysSock2SetOption(socket, SysSocket2.GVL.SOCKET_SOL, SysSocket2.GVL.SOCKET_SO_REUSEADDR, ADR(dint_true), SIZEOF(dint_true));
		// Set option for keepalive
		//FunctionResult := SysSock2SetOption(socket, SOCKET_SOL, SOCKET_SO_KEEPALIVE, ADR(dint_true), SIZEOF(dint_true));
		IF TLS THEN
			FunctionResult := SysSocket2.SysSock2Ioctl(socket, SysSocket2.GVL.SOCKET_FIONBIO, ADR(dint_false)); (* Blocking mode for connect to TLS*)
		ELSE
        	FunctionResult := SysSocket2.SysSock2Ioctl(socket, SysSocket2.GVL.SOCKET_FIONBIO, ADR(dint_true)); (* NonBlocking mode *)
		END_IF
		sockaddr.sin_family := SysSocket2.GVL.SOCKET_AF_INET;
		sockaddr.sin_port := SysSocket2.SysSock2Ntohs(c_port);
		sockaddr.sin_addr.ulAddr  := SysSocket2.SysSock2Ntohl(c_ip);
		c_select := FALSE;
		state := TC_CONNECT;
	END_IF;

(* ---------------------------------------------- *)

TC_CONNECT:
	IF NOT c_enable OR c_status = 255 THEN (* keine freigabe oder connect timeout *)
			state:= C_CLOSE;
	ELSE
		IF c_select = FALSE THEN
			TlsConnectLastTick := OSCAT_BASIC.T_PLC_MS();
			{info 'TODO: hind that this is blocking!'}
			pResult:=SysSocket2.SysSock2Connect(socket,ADR(sockaddr),SIZEOF(sockaddr));
			TlsConnectTime := OSCAT_BASIC.T_PLC_MS() - TlsConnectLastTick; 
			IF pResult = CmpErrors.Errors.ERR_OK OR pResult =  CmpErrors.Errors.ERR_SOCK_ISCONNECTED THEN 
				c_ready := TRUE; (* Connected *)
				state:= C_WAIT;
				IF TLS THEN
        			SysSocket2.SysSock2Ioctl(socket,SysSocket2.GVL.SOCKET_FIONBIO, ADR(dint_true)); (* NonBlocking mode *)
				END_IF
			ELSE
				IF tls THEN
					state:= C_CLOSE;//TLS connect ist blokierend, wenn hier, fehler, reset 
				ELSE
					(* Connect durchgeführt, aber noch nicht verbunden, dann optional mit select-abfrage weitermachen *)
					c_select := OSCAT_NETWORK_TYPES.SYSLIBSOCKETS_OPTION.0; (* Bit 0 = TCP-Client - use SysSock2select *)
				END_IF
				//c_select := TRUE;
			END_IF;

		
		ELSE
			c_Timeout.tv_sec := 0;
			c_Timeout.tv_usec := 0;
			c_fdWrite.fd_count := 1;
			c_fdWrite.fd_array[0] := socket;
			//IF SysSock2Select(SOCKET_FD_SETSIZE,0,ADR(c_fdWrite),0, ADR(c_Timeout), ADR(pResult)) > 0 THEN
			IF SysSocket2.SysSock2Select(
				hSocket:= socket, 
				diWidth:= SysSocket2.GVL.SOCKET_FD_SETSIZE, 
				pfdRead:= 0, 
				pfdWrite:= ADR(c_fdWrite), 
				pfdExcept:= 0, 
				ptvTimeout:= ADR(c_Timeout), 
				pdiReady:= ADR(pResult)) > 0 THEN
				c_ready := TRUE; (* Connected *)
				state:= C_WAIT;
				IF TLS THEN
        			FunctionResult := SysSocket2.SysSock2Ioctl(socket, SysSocket2.GVL.SOCKET_FIONBIO, ADR(dint_true)); (* NonBlocking mode *)
				END_IF
			END_IF;
		END_IF;
	END_IF;

(* ---------------------------------------------- *)

TS_INIT: (* TCP-SERVER (PASSIV) *)
	//	server_socket := SysSock2Create(SOCKET_AF_INET, SOCKET_STREAM, SOCKET_IPPROTO_IP, ADR(pResult)); (* Create Socket *)
	SysSockParameter.parameterType := SysSocket2.SysSocket2_Type.STD;
	SysSockSpec.stdSockets.i32AddressFamily := SysSocket2.GVL.SOCKET_AF_INET;
	SysSockSpec.stdSockets.i32Type := SysSocket2.GVL.SOCKET_STREAM;
	SysSockSpec.stdSockets.i32Protocol := SysSocket2.GVL.SOCKET_IPPROTO_IP;
	SysSockParameter.specific := SysSockSpec;
	server_socket := SysSocket2.SysSock2Create(pParameter:= ADR(SysSockParameter), pResult:= ADR(pResult));
	
	IF server_socket = SysTypes.RTS_INVALID_HANDLE THEN
		c_status := 1; (* SysSock2Create failed *)
		state:= C_CLOSE;
	ELSE (* Address bindings *)
		SysSocket2.SysSock2SetOption( server_socket, SysSocket2.GVL.SOCKET_SOL, SysSocket2.GVL.SOCKET_SO_REUSEADDR, ADR(dint_true), SIZEOF(dint_true) );
		sockaddr.sin_family:= SysSocket2.GVL.SOCKET_AF_INET;
		sockaddr.sin_port := SysSocket2.SysSock2Htons(c_port);
		sockaddr.sin_addr.ulAddr  := SysSocket2.GVL.SOCKET_INADDR_ANY;
		IF NOT SysSocket2.SysSock2Bind(server_socket, ADR(sockaddr), SIZEOF(sockaddr)) = 0 THEN
			c_status := 2; (* SysSock2Bind failed *)
			state := C_CLOSE;
		ELSIF NOT SysSocket2.SysSock2Listen(server_socket, 1) = 0 THEN (* erzeugt Warteschlange für eine Verbindung *)
			c_status := 3; (* SysSock2Listen failed *)
			state:= C_CLOSE;
		ELSE
			SysSocket2.SysSock2Ioctl(server_socket, SysSocket2.GVL.SOCKET_FIONBIO, ADR(dint_true)); (* NonBlocking mode *)
			state:= TS_OPEN;
		END_IF;
	END_IF;

(* ---------------------------------------------- *)

TS_OPEN: (* Waiting for incomming connection *)
	sockaddr_size := SIZEOF(sockaddr);
	socket := SysSocket2.SysSock2Accept(server_socket, ADR(sockaddr), ADR(sockaddr_size), ADR(pResult));

	IF socket <> SysTypes.RTS_INVALID_HANDLE THEN (* neuer Verbindungswunsch vorhanden *)
		IF c_mode = BYTE#2 AND sockaddr.sin_addr.ulAddr <> SysSocket2.SysSock2Ntohl(c_ip) THEN (* Mode 2 = TCP + PASSIVE + PORT + IP  auf richtige Partner-IP prüfen *)
			state:= C_CLOSE;
		ELSE
			IF plc_841 OR plc_881 THEN
				SysSocket2.SysSock2SetOption(socket, 6, SysSocket2.GVL.SOCKET_TCP_NODELAY, ADR(dint_true), SIZEOF(dint_true)); (* Set Push-Bit *)
			END_IF;
			SysSocket2.SysSock2Ioctl(socket, SysSocket2.GVL.SOCKET_FIONBIO, ADR(dint_true)); (* NonBlocking mode *)
			c_ready := TRUE; (* Connected *)
			state := C_WAIT;
		END_IF;
	ELSIF NOT c_enable THEN (* keine freigabe mehr ? *)
			state:= C_CLOSE;
	END_IF;

(* ---------------------------------------------- *)

C_WAIT: (* Warten auf Anforderung für Beenden *)
	IF NOT c_enable OR NOT c_ready THEN
		state:= C_CLOSE;
	END_IF

(* ---------------------------------------------- *)

C_CLOSE: (* Close the Sockets *)
	c_ready := FALSE;
	IF socket >= 0 THEN
		IF (NOT plc_841) AND (NOT plc_881) THEN
			IF udp_mode THEN
				SysSocket.SysSockShutdown(socket, 0);
			ELSE
				SysSocket2.SysSock2Shutdown(socket, 0); (* 870 *)
			END_IF
		END_IF;
		IF udp_mode THEN
			pResult := SysSocket.SysSockClose(socket);
		ELSE
			pResult := SysSocket2.SysSock2Close(socket);	
		END_IF
		IF TLS THEN
			// cleanup TLS Context
			CmpTls.CmpTlsFreeContext(hTlsContext:= SysSockSpec.tlsSockets.hTlsContext);
		END_IF
		socket := SysTypes.RTS_INVALID_HANDLE;
		SysSockSpec.tlsSockets.hTlsContext := SysTypes.RTS_INVALID_HANDLE; 
	END_IF
	IF server_socket >= 0 THEN
		IF (NOT plc_841) AND (NOT plc_881) THEN
			SysSocket2.SysSock2Shutdown(server_socket, 0); (* 870 *)
		END_IF;
		SysSocket2.SysSock2Close(server_socket);
		server_socket := SysTypes.RTS_INVALID_HANDLE;
	END_IF
	state:= STOP;
END_CASE;

(* ---------------------------------------------- *)

IF c_ready THEN
	IF NOT c_ready_old THEN (* Verbindung aufgebaut - positive Flanke erkannt *)
		IP_C.C_STATE := 254;
		IP_C.TIME_RESET := TRUE; (* Alle Timer ruecksetzen *)
		(* ---------------------- Debug-Message ----------------------------*)
		(*IF _debug_enable THEN
			LOG_CL.NEW_MSG := 'IP_CON: CONNECTED -IP_ID ~6';
			LOG_CL.PRINTF[6] := INT_TO_STRING(debug_ID);
			LOG_MSG();
		END_IF;*)
		(* -----------------------------------------------------------------------------*)
	ELSE
		IP_C.C_STATE := 255; (* Verbindung ist aufgebaut *)
	END_IF;
ELSE
	IF c_ready_old THEN (* Verbindung abgebaut - negative Flanke erkannt *)
		IP_C.C_STATE := 1;
		IP_C.MAILBOX[1] := 0; (* Receive Info rücksetzen *)
		IP_C.MAILBOX[2] := 0; (* Send-Pause rücksetzen *)
		IP_C.MAILBOX[3] := 0; (* Receive-Pause rücksetzen *)
		IF NOT new_connection THEN
			s_active := FALSE; (* Sendeaktivitäten stoppen *)
			s_req := FALSE; (* Sendefreigabe rücksetzen *)
			S_BUF.SIZE := 0; (* Sendelänge löschen *)
			(*IP_C.TIME_RESET := TRUE;*) (* Alle Timer ruecksetzen *)
		END_IF;
		(* ---------------------- Debug-Message ----------------------------*)
		(*IF _debug_enable THEN
			LOG_CL.NEW_MSG := 'IP_CON: DISCONNECTED';
			LOG_MSG();
		END_IF;*)
		(* -----------------------------------------------------------------------------*)
	ELSE
		IP_C.C_STATE := 0; (* Verbindung ist abgebaut *)
	END_IF;
END_IF;

c_ready_old := c_ready;

(* Der Datenempfang wird angehalten solange ein Sendevorgang läuft *)
(* sonst kann es vorkommen das die Antwort-daten schon empfangen werden, *)
(* bevor der Sendevorgang vom programm abgeschlossen wurde *)

IF c_ready AND NOT s_active AND IP_C.MAILBOX[3] = 0 THEN
	IF R_BUF.SIZE >= INT_TO_UINT(r_max_size) THEN
		R_BUF.SIZE := UINT#0;
		r_status := 254; (* Empfangsbuffer wegen Überlauf rückgesetzt *)
	END_IF;

	r_offset := SEL(udp_mode,UINT_TO_INT(R_BUF.SIZE),0);
	r_count := r_max_size - r_offset;

	IF udp_mode THEN

		bytes_received := TO_DINT(SysSocket.SysSockRecvFrom(socket, ADR(R_BUF.BUFFER), r_count, 0, ADR(sockaddrUDP), SIZEOF(sockaddrUDP), ADR(pResult)));
		IF c_mode = BYTE#3 AND sockaddrUDP.sin_addr.ulAddr <> SysSocket.SysSockNtohl(c_ip) THEN (* Mode 3 = UDP + PASSIVE + PORT + IP  auf richtige Partner-IP prüfen *)
			bytes_received := 0;
			R_BUF.SIZE := UINT#0;
			sockaddrUDP.sin_port := SysSocket.SysSockNtohs(c_port);
			sockaddrUDP.sin_addr.ulAddr  := SysSocket.SysSockNtohl(c_ip);
		END_IF;

	ELSE
		bytes_received := TO_DINT(SysSocket2.SysSock2Recv(socket, ADR(R_BUF.BUFFER[r_offset]), r_count, 0, ADR(pResult)));
	END_IF;

	CASE pResult OF
		518:  bytes_received:=-1; //Connection OKAY just no data and do not want to BIND
		521:  bytes_received:=0; //Connection has been refused by the remote host 
		523:  bytes_received:=0; //The host has not been found  
		524:  bytes_received:=0; //Host is unreachable  
		526:  bytes_received:=0; //The socket is not connected  
		527:  bytes_received:=0; //Shutdown has been called on the socket  
		529:  bytes_received:=0; //Socket has been gracefully closed. No more send/receives allowed	 
	END_CASE

	
	(*UDP: IPC returns -1 if no data available or error occured,841 returns -1 if error occured and 0 if no data available*)
	CASE bytes_received OF
	-2147483648..-1: ; (* No data available or error occured *)
	 0: IF NOT udp_mode OR pResult<>518 THEN (* TCP-Mode: socket wurde von remote geschlossen *)
			c_status := 253;
			c_ready := FALSE;
			IP_C.ResultReceive := pResult;
		END_IF;
	ELSE (* daten wurden empfangen *)
  		r_time := tx; (* Receive Timer ruecksetzen *)
		R_BUF.SIZE := INT_TO_UINT(r_offset) + DINT_TO_UINT(bytes_received); (* aktuelle buffersize eintragen *)
		IP_C.MAILBOX[1] := IP_C.MAILBOX[1] + 1; (* Receive Info *)
		IF IP_C.MAILBOX[1] = 0 THEN IP_C.MAILBOX[1] := 1; END_IF;

		(* ---------------------- Debug-Message ----------------------------*)
		(*IF _debug_enable THEN
			LOG_CL.NEW_MSG := 'IP_REC DATA: POS: ~1 : SIZE: ~2 TOTAL ~3 -IP_ID ~6';
			LOG_CL.PRINTF[1] := INT_TO_STRING(r_offset);
			LOG_CL.PRINTF[2] := INT_TO_STRING(r_count);
			LOG_CL.PRINTF[3] := UINT_TO_STRING(R_BUF.SIZE);
			LOG_CL.PRINTF[6] := INT_TO_STRING(debug_ID);
			LOG_MSG();
		END_IF;*)
		(* -----------------------------------------------------------------------------*)

	END_CASE
END_IF;

(* ---------------------------------------------- *)

IF S_BUF.SIZE > 0 THEN
	IF c_ready AND c_enable THEN
		IF NOT s_active AND IP_C.MAILBOX[2] = 0 THEN
			(* Gesamtanzahl an Bytes limitieren und uebergeben *)
			s_total := LIMIT(0,UINT_TO_INT(S_BUF.SIZE),r_max_size);
			s_cur_pos  := 0;
			s_cur_size := 0;
			s_start := TRUE; (* Daten kopieren und senden anstossen *)
			s_active := TRUE; (* Sende-Betrieb aktivieren *)
			(* ---------------------- Debug-Message ----------------------------*)
			(*IF _debug_enable THEN
				LOG_CL.NEW_MSG := 'IP_SEN INIT: TOTAL: ~1 -IP_ID ~6';
				LOG_CL.PRINTF[1] := INT_TO_STRING(S_TOTAL);
				LOG_CL.PRINTF[6] := INT_TO_STRING(debug_ID);
				LOG_MSG();
			END_IF;*)
			(* -----------------------------------------------------------------------------*)
		END_IF;

		IF s_done OR s_start THEN (* Daten senden aktiv *)

			s_start := FALSE;
			s_cur_pos := s_cur_pos + s_cur_size; (* neue Sende-Datenposition bestimmen *)
			IF s_total > s_cur_pos THEN (* weitere Daten zum senden vorhanden ? *)
				s_cur_size := s_total - s_cur_pos;
				s_cur_size := LIMIT(0, s_cur_size, s_max_size); (* Telegrammlänge begrenzen *)
				(* ---------------------- Debug-Message ----------------------------*)
				(*IF _debug_enable THEN
					LOG_CL.NEW_MSG := 'IP_SEN DATA: POS: ~1 : SIZE: ~2 TOTAL ~3 -IP_ID ~6';
					LOG_CL.PRINTF[1] := INT_TO_STRING(S_CUR_POS);
					LOG_CL.PRINTF[2] := INT_TO_STRING(S_CUR_SIZE);
					LOG_CL.PRINTF[3] := INT_TO_STRING(S_TOTAL);
					LOG_CL.PRINTF[6] := INT_TO_STRING(debug_ID);
					LOG_MSG();
				END_IF;*)
				(* -----------------------------------------------------------------------------*)
				s_time := tx; (* Send Timer ruecksetzen *)
				r_time := tx; (* Receive Timer ruecksetzen *)
				s_req := TRUE;

			ELSE
				(* keine weitere Sendedaten vorhanden -> Senden beenden *)
				s_req := FALSE;
				s_active := FALSE;
				S_BUF.SIZE := 0;
				(* ---------------------- Debug-Message ----------------------------*)
				(*IF _debug_enable THEN
					LOG_CL.NEW_MSG := 'IP_SEN FINISH -IP_ID ~6';
					LOG_CL.PRINTF[6] := INT_TO_STRING(debug_ID);
					LOG_MSG();
				END_IF;*)
				(* -----------------------------------------------------------------------------*)
			END_IF;
		END_IF;
	END_IF;
END_IF;

IF s_req THEN
	s_done := FALSE;
	IF udp_mode THEN
		bytes_sent := TO_DINT(SysSocket.SysSockSendTo(socket, ADR(S_BUF.BUFFER[s_cur_pos]), s_cur_size, 0, ADR(sockaddr), SIZEOF(sockaddr), ADR(pResult)));
	ELSE
		bytes_sent := TO_DINT(SysSocket2.SysSock2Send(socket, ADR(S_BUF.BUFFER[s_cur_pos]), s_cur_size, 0, ADR(pResult)));
	END_IF;

	CASE bytes_sent OF
	-2147483648..-1:	; (* ERROR: Noch nicht bereit um Daten aufzunehmen -> nächsten Zyklus wieder probieren *)
	 0: IF NOT udp_mode AND pResult<>518 THEN (* TCP-Mode: socket wurde von remote geschlossen *)
			c_status := 253;
			c_ready := FALSE;
			IP_C.ResultSend := pResult;
		END_IF;
	ELSE
		s_done := TRUE;
		s_cur_size := DINT_TO_INT(bytes_sent); (* Anzahl der wirklich versendeten Bytes übernehmen *)
		(* ---------------------- Debug-Message ----------------------------*)
		(*IF _debug_enable THEN
			LOG_CL.NEW_MSG := 'IP_SEN SEND_COUNT ~1 -IP_ID ~6';
			LOG_CL.PRINTF[1] := DINT_TO_STRING(s_cur_size);
			LOG_CL.PRINTF[6] := INT_TO_STRING(debug_ID);
			LOG_MSG();
		END_IF;*)
		(* -----------------------------------------------------------------------------*)
	END_CASE
END_IF;

(* ---------------------------------------------- *)

IF IP_C.R_OBSERVE = FALSE OR s_active THEN
    r_time := tx;
END_IF;

IF c_status = 0 AND tx - c_time > error_time AND c_enable AND NOT c_ready AND c_mode < 2 THEN (* Connect Timeout *)
	c_status := 255; (* Timeout-Fehler ausgeben *)
END_IF;
IF s_status = 0 AND tx - s_time > error_time AND s_active THEN (* Send Timeout *)
	s_status := 255; (* Timeout-Fehler ausgeben *)
END_IF;
IF r_status = 0 AND tx - r_time > error_time AND c_ready AND IP_C.R_OBSERVE THEN (* Receive Timeout *)
	r_status := 255; (* Timeout-Fehler ausgeben *)
END_IF;

IP_C.ERROR := OSCAT_BASIC.DWORD_OF_BYTE(c_status,s_status,r_status,0);

(* ---------------------- Debug-Message ----------------------------*)
(*IF  _debug_enable THEN
	IF (IP_C.ERROR <> debug_lasterror) THEN
		LOG_CL.NEW_MSG := 'IP_ERROR ~1 -IP_ID ~6';
		LOG_CL.PRINTF[1] := DWORD_TO_STRING(IP_C.ERROR);
		LOG_CL.PRINTF[6] := INT_TO_STRING(debug_ID);
		LOG_MSG();

		debug_lasterror := IP_C.ERROR;
		debug_last_id := debug_ID;
	END_IF;
END_IF;*)
(* -----------------------------------------------------------------------------*)

(* revision history
ks	18. oct. 2008	rev 1.0
	original version
ks	05. jan. 2009	rev 1.1
	zusätzlichen Parameter "Port" hinzugefügt, und Code bei Verbindungsaufbau angepasst
ks	28. feb. 2009	rev 1.2
	connect code angepasst und verkürzung der zyklen bei Send
ks	20. oct. 2009	rev 1.3
	network_buffer basis 0
ks	06. dec. 2009	rev 1.4
	receive_count MAILBOX[1]
ks	10. nov. 2010	rev 1.5
	send_pause MAILBOX[2] and receive_pause MAILBOX[3] 
ks	07. feb. 2011	rev 1.6
	Fehlercode 253 bei Remote-Verbindungsabbruch
ks	30. may. 2011	rev 1.7
	Fehler bei Empfangsüberwachung
ks	26. july. 2011	rev 1.8
	Error-Reset, diverse optimierungen 
ks	26. feb. 2012	rev 1.9
	Code-Optimierung für höhere kompatibilität

*)

END_FUNCTION_BLOCK

// Common/Function Blocks/TIME_DATE_IMPULS
FUNCTION_BLOCK TIME_DATE_IMPULS
VAR_IN_OUT
	TDI_Data:TIME_DATE_IMPULS_DATA;
END_VAR
VAR_INPUT
END_VAR

VAR
	RT_SYS:Time_and_Date.RTCLK.GetDateAndTime;
	RT:OSCAT_BASIC.RTC_2;
	DT_OLD:DT;
	GET_TIME: BOOL := TRUE;
	TIME_READED: BOOL;
	TIMEZONE:Time_and_Date.RTCLK.PERIODE;
	ReReadTime: BOOL;
	ReReadErrorTime:TON;
	ReReadTimeCycle:TON;
	DayChangeEdge:R_TRIG;
END_VAR

RT_SYS(xExecute := GET_TIME);
IF RT_SYS.xDone THEN
	GET_TIME := FALSE;
	IF	RT_SYS.dtDateAndTime < DT#1980-01-01-00:00:00 THEN
		//Keine Valide Uhr auf Raspi!
		ReReadTime := TRUE;
		TDI_Data.TIME_IO := FALSE;
	ELSE
		TIME_READED := TRUE;
		TIMEZONE := RT_SYS.eTimezone;
		ReReadTime := FALSE;
		TDI_Data.TIME_IO := TRUE;
	END_IF
END_IF
//Zykliches neulsesen der Uhrzeit
ReReadTimeCycle(in := (TDI_Data.TIME_IO AND NOT GET_TIME), PT:= T#30M);
IF ReReadTimeCycle.Q THEN
	GET_TIME := TRUE;//try again to read Time	
END_IF


//Neulesezeit nach Error bearbeiten:
ReReadErrorTime(in:=ReReadTime, pt:=T#1S);
IF ReReadErrorTime.Q THEN
	ReReadTime := FALSE;
	GET_TIME := TRUE;//try again to read Time
END_IF
//Realtime Clock bearbeiten // Setzten
RT(set := TIME_READED, SDT := RT_SYS.dtDateAndTime, OFS := 60, DEN:=TRUE,);
TIME_READED := FALSE;
//Date and time from oscat fb
TDI_Data.SYSTEM_TIME:=RT.LOCAL_DT;
//check for second impuls
IF DT_OLD <> TDI_Data.SYSTEM_TIME THEN
	DT_OLD := TDI_Data.SYSTEM_TIME;
	TDI_Data.imp := TRUE;
ELSE
	TDI_Data.imp := FALSE;
END_IF
//make Time for OSCAT functions
TDI_Data.TD_TIME := OSCAT_BASIC.DT_TO_SDT(DTI:= TDI_Data.SYSTEM_TIME);
TDI_Data.UDT := RT.UDT;

DayChangeEdge(CLK:=TO_TOD(TDI_DATA.SYSTEM_TIME)= TOD#00:00:00);
TDI_DATA.DAY_CHANGE := DayChangeEdge.Q;

END_FUNCTION_BLOCK

// Common/Functions/GET_DNS_IP
FUNCTION GET_DNS_IP : STRING(16)
VAR_INPUT
END_VAR
VAR
	Result:SysTypes.RTS_IEC_RESULT;
	DNS_STRING:STRING(1000);
	findRet:DINT;
	i:INT;
	j:INT;
	k:INT;
	start:INT;
	stop:INT;
	//id of operating system
	OsId:UDINT;
END_VAR
VAR CONSTANT
	GET_DNS_COMMAND_LINUX:STRING:='cat /etc/resolv.conf ';//|grep -i nameserver|head -n1|cut -d $' $' -f2';
	GET_DNS_COMMAND_WINDOWS:STRING:='powershell Get-DnsClientServerAddress';//|grep -i nameserver|head -n1|cut -d $' $' -f2';
	NAMESERVER_LINUX:STRING:='nameserver';
	
END_VAR

(*
for linux

change 
sudo nano /etc/CODESYSControl.cfg
or from runtime version 4.5.11.20
sudo nano /etc/CODESYSControl_User.cfg 
[SysProcess]
Command.0=shutdown

to 

[SysProcess]
Command.0=shutdown
Command.1=cat

for windows, needs powershell

"C:\ProgramData\CODESYS\CODESYSControlWinV3\???\CODESYSControl.cfg"
[SysProcess]
BasePriority=Realtime
Command=AllowAll

*)

//cat /etc/resolv.conf |grep -i nameserver|head -n1|cut -d ' ' -f2
//get content

SysTarget.SysTargetGetOperatingSystemId(pudiOperatingSystemId:= ADR(OsId));


GET_DNS_IP := 'ERROR';

IF OsId = SysTarget.OperatingSystemID.SYSTARGET_OS_LINUX THEN

	SysProcess.SysProcessExecuteCommand2(pszCommand:=GET_DNS_COMMAND_LINUX,pszStdOut:= DNS_STRING,udiStdOutLen:=SIZEOF(DNS_STRING),pResult:=ADR(Result));
	IF Result = CmpErrors.Errors.ERR_NO_ACCESS_RIGHTS THEN
		GET_DNS_IP := 'NOACCESSRIGHTS';
		RETURN;
	END_IF
	//TODO check if command is enabled 
	i:= Standard.FIND(STR1:=DNS_STRING, STR2:=NAMESERVER_LINUX);
	IF i < 0 THEN RETURN; END_IF
	j := OSCAT_BASIC.FIND_CTRL(str:= DNS_STRING, pos:= i);
	IF j <= 0 THEN RETURN; END_IF
	
	GET_DNS_IP := Standard.MID(STR:= DNS_STRING, LEN:= j - i - Standard.LEN(STR:=NAMESERVER_LINUX) - 1, POS:= i + Standard.LEN(NAMESERVER_LINUX) + 1);
	
END_IF

IF OsId = SysTarget.OperatingSystemID.SYSTARGET_OS_WINDOWS THEN
{info 'TODO: hind that this is blocking!'}
SysProcess.SysProcessExecuteCommand2(pszCommand:=GET_DNS_COMMAND_WINDOWS,pszStdOut:= DNS_STRING,udiStdOutLen:=SIZEOF(DNS_STRING),pResult:=ADR(Result));
	IF Result = CmpErrors.Errors.ERR_NO_ACCESS_RIGHTS THEN
		GET_DNS_IP := 'NOACCESSRIGHTS';
		RETURN;
	END_IF
	//TODO check if command is enabled 
	findRet:= find(STR1:=ADR(DNS_STRING), STR2:=ADR('IPv4'));
	IF findRet < 0 THEN RETURN; END_IF
	i := DINT_TO_INT(findRet);
	//now search '{'
	FOR j := 0 TO 40 DO//max 40 chars space
		IF DNS_STRING[i + j] = GetChar('{') THEN
			start := i + j + 1;
		END_IF
 		IF DNS_STRING[i + j] = GetChar('}') THEN
			stop := i + j - 1;
			EXIT;
		END_IF
	END_FOR
	//now copy data, string functions usless --> more than 255 chars...
	
	j := 0;
	FOR i := start TO stop DO
		GET_DNS_IP[j] := DNS_STRING[i];
		j := j + 1;
	END_FOR
	GET_DNS_IP[j] := 0;//termination
	
	//j := OSCAT_BASIC.FIND_CTRL(str:= DNS_STRING, pos:= i);
//	IF j <= 0 THEN RETURN; END_IF
	
	//GET_DNS_IP := Standard.MID(STR:= DNS_STRING, LEN:= j - i - Standard.LEN(STR:=NAMESERVER_LINUX) - 1, POS:= i + Standard.LEN(NAMESERVER_LINUX) + 1);
	

END_IF

END_FUNCTION

// Common/Functions/find
//searchs str2 in str1
FUNCTION find : DINT
VAR_INPUT
	str1:POINTER TO STRING;
	str2:POINTER TO STRING;
END_VAR
VAR
	
	n:UINT;	
	pt:POINTER TO BYTE;
	
	j: UINT;
END_VAR

find := -1;//first we din't find anything....
n := len(str := str2);


pt := str1;

WHILE pt^ <> 0 DO
	IF SysMem.SysMemCmp(pBuffer1:= pt, pBuffer2:= str2, udiCount:= n) = 0 THEN
		
		find := j;
		RETURN;
	
	END_IF
	j := j + 1;
	pt := pt + SIZEOF(BYTE);
	
END_WHILE

END_FUNCTION

// Common/Functions/len
FUNCTION len : UINT
VAR_INPUT
	str:POINTER TO STRING;
END_VAR
VAR
	k:uINT;
	pt:POINTER TO BYTE;
END_VAR

pt := str;
WHILE pt[k] <>  0 DO
	k := k + 1;
END_WHILE
len := k;

END_FUNCTION

// Common/Functions/GetChar
FUNCTION GetChar : byte
VAR_INPUT
	in:STRING(1);
END_VAR

GetChar := in[0];

END_FUNCTION

// Common/Functions/concat
FUNCTION concat : pointer to string
VAR_INPUT
	s1:POINTER TO STRING;
	s2:POINTER TO STRING;
END_VAR
VAR
	p1:POINTER TO BYTE;
	len1:UINT;
	
	ui:UINT;
END_VAR

p1 := ADR(s1^[len(s1)]);
len1 := len(s2);
SysMem.SysMemMove(pDest:= p1, pSrc:= s2, udiCount:= len1 + 1);//+ 1 for add 0 to string end

concat := s1;

END_FUNCTION

// Common/Function Blocks/TestString
FUNCTION_BLOCK TestString 
VAR_INPUT
END_VAR
VAR
	s10:STRING:='1111111111';
	s102:STRING:='2222222222';
	sp:STRING(64000);
	ps1:POINTER TO STRING;
	lens:UINT;
END_VAR

lens := len(ADR(s10)); //needs to be 10!
sp:='';
concat(s1:= ADR(sp), s2:= ADR(s10));
ps1 := ADR(sp);
lens := len(ADR(sp)); //needs to be 10!

concat(s1:= ADR(sp), s2:= ADR(s102));

lens := len(ADR(sp)); //needs to be 20!

concat(s1:= ADR(sp), s2:= ADR(s10));

lens := len(ADR(sp)); //needs to be 30!

concat(s1:= ADR(sp), s2:= ADR(s102));

lens := len(ADR(sp)); //needs to be 40!

concat(s1:= ADR(sp), s2:= ADR(s10));

lens := len(ADR(sp)); //needs to be 50!

concat(s1:= ADR(sp), s2:= ADR(sp));

lens := len(ADR(sp)); //needs to be 100!

concat(s1:= ADR(sp), s2:= ADR(sp));

lens := len(ADR(sp)); //needs to be 200!

concat(s1:= ADR(sp), s2:= ADR(sp));

lens := len(ADR(sp)); //needs to be 400!

concat(s1:= ADR(sp), s2:= ADR(sp));

lens := len(ADR(sp)); //needs to be 800!

concat(s1:= ADR(sp), s2:= ADR(sp));

lens := len(ADR(sp)); //needs to be 1600!

concat(s1:= ADR(sp), s2:= ADR(sp));

lens := len(ADR(sp)); //needs to be 3200!

concat(s1:= ADR(sp), s2:= ADR(sp));

lens := len(ADR(sp)); //needs to be 6400!

END_FUNCTION_BLOCK

// Common/Function Blocks/IP_CONTROL_TLS
FUNCTION_BLOCK IP_CONTROL_TLS EXTENDS IP_CONTROL
VAR_INPUT
	TLS_CONFIG_IN:POINTER TO TLS_CONFIG := 0;(*info about tls stuff*)
	useTls: BOOL;

END_VAR
VAR_OUTPUT
END_VAR
VAR
	
END_VAR


TLS:= useTls;
IF TLS THEN
	TLS_CONFIG := TLS_CONFIG_IN;
END_IF
//SUPER^();
SUPER^(IP_C := IP_C, R_BUF:= R_BUF, S_BUF:= S_BUF, IP:= IP, PORT:= PORT, TIME_OUT:= TIME_OUT);

END_FUNCTION_BLOCK

// Common/Functions/ResolveIPAddr
/// This function resolves the IP of the domain name. 
FUNCTION ResolveIPAddr : SysTypes.RTS_IEC_RESULT
VAR_INPUT
	sHost : STRING;
	sIPResult : POINTER TO STRING; 
END_VAR
VAR
	refsHost : REFERENCE TO STRING := sHost;
	stSockHost : SysSocket.SOCK_HOSTENT;
	rtsResultSock : SysTypes.RTS_IEC_RESULT;
	rtsResultInAddr : SysTypes.RTS_IEC_RESULT;
	stinAddr : SysSocket.INADDR;
	ptdwHostAddr : POINTER TO __XWORD;
	dwHostAddr : __XWORD;
	sServerIP : STRING;
END_VAR

rtsResultSock := SysSocket.SysSockGetHostByName(refsHost,ADR(stSockHost));
IF rtsResultSock = CmpErrors.Errors.ERR_OK THEN
	ptdwHostAddr := stSockHost.pAddrList[0]; // Eth Adapter
	dwHostAddr := ptdwHostAddr^;
	IF dwHostAddr <> SysSocket.GVL.SOCKET_INADDR_NONE THEN
		stinAddr.ulAddr := __XWORD_TO_UDINT(dwHostAddr);
		rtsResultInAddr := SysSocket.SysSockInetNtoa(pInAddr:=ADR(stinAddr),szIPADDR:=sServerIP ,diIPAddrSize:=SIZEOF(sServerIP));
		IF rtsResultInAddr = CmpErrors.Errors.ERR_OK THEN
			sIPResult^ := sServerIP;
		ELSE
			ResolveIPAddr := CmpErrors.Errors.ERR_FAILED;
		END_IF
	END_IF
ELSE
	ResolveIPAddr := CmpErrors.Errors.ERR_FAILED;
END_IF

END_FUNCTION

// Common/Functions/CheckDeltaValue
FUNCTION CheckDeltaValue : bool
VAR_INPUT
	Value:ALL_TYPES_UNION;
	TypeOfValue:IBaseLibrary.TypeClass;
	//TypeOfValue:VAR_TYPES;
	DeltaVar:UINT;
	Faktor:UINT;
END_VAR
VAR_IN_OUT
	LastValue:ALL_TYPES_UNION;
END_VAR
VAR
END_VAR

(*	SINT_T, USINT_T, INT_T, UINT_T, DINT_T, UDINT_T, 
				LINT_T, ULINT_T, REALT_T, LREAL_T*)
CASE TypeOfValue OF
	IBaseLibrary.TypeClass.TYPE_BOOL:
		CheckDeltaValue := LastValue.BOOL_T <> Value.BOOL_T;
		IF CheckDeltaValue THEN LastValue.BOOL_T := Value.BOOL_T; END_IF
	IBaseLibrary.TypeClass.TYPE_SINT:
	//VAR_TYPES.SINT_T:
		//CheckDeltaValue := (ABS(LAST_VALUE.SINT_T) + UINT_TO_SINT(DELTA_VAR)) > ABS(Value.SINT_T);
		CheckDeltaValue := ABS(LastValue.SINT_T - Value.SINT_T) >= UINT_TO_SINT(DeltaVar);
		IF CheckDeltaValue THEN LastValue.SINT_T := Value.SINT_T; END_IF
	//VAR_TYPES.USINT_T:
	IBaseLibrary.TypeClass.TYPE_USINT:
		CheckDeltaValue := ABS(USINT_TO_INT(LastValue.USINT_T) - USINT_TO_INT(Value.USINT_T)) >= UINT_TO_USINT(DeltaVar);
		IF CheckDeltaValue THEN LastValue.USINT_T := Value.USINT_T; END_IF
	//VAR_TYPES.INT_T:
	IBaseLibrary.TypeClass.TYPE_INT:
		CheckDeltaValue := ABS(LastValue.INT_T - Value.INT_T) >= + UINT_TO_INT(DeltaVar);
		IF CheckDeltaValue THEN LastValue.INT_T := Value.INT_T; END_IF
	//VAR_TYPES.UINT_T:
	IBaseLibrary.TypeClass.TYPE_UINT:
		CheckDeltaValue := ABS(UINT_TO_DINT(LastValue.UINT_T) - UINT_TO_DINT(Value.UINT_T)) >= DeltaVar;
		IF CheckDeltaValue THEN LastValue.UINT_T := Value.UINT_T; END_IF
	//VAR_TYPES.DINT_T:
	IBaseLibrary.TypeClass.TYPE_DINT:
		CheckDeltaValue := ABS(LastValue.DINT_T - Value.DINT_T) >= + UINT_TO_DINT(DeltaVar);
		IF CheckDeltaValue THEN LastValue.DINT_T := Value.DINT_T; END_IF
	//VAR_TYPES.UDINT_T:
	IBaseLibrary.TypeClass.TYPE_UDINT:
		CheckDeltaValue := ABS(UDINT_TO_LINT(LastValue.UDINT_T) - UDINT_TO_LINT(Value.UDINT_T)) >= DeltaVar;
		IF CheckDeltaValue THEN LastValue.UDINT_T := Value.UDINT_T; END_IF
	//VAR_TYPES.LINT_T:
	IBaseLibrary.TypeClass.TYPE_LINT:
		CheckDeltaValue := ABS(LastValue.LINT_T - Value.LINT_T) >= + UINT_TO_LINT(DeltaVar);
		IF CheckDeltaValue THEN LastValue.LINT_T := Value.LINT_T; END_IF
	//VAR_TYPES.ULINT_T:
	IBaseLibrary.TypeClass.TYPE_ULINT:
	//here we use no expand but check min max because no bigger data type...
		IF LastValue.ULINT_T <= Value.ULINT_T THEN
			CheckDeltaValue := Value.ULINT_T - LastValue.ULINT_T >= UINT_TO_ULINT(DeltaVar);	
		ELSE
			CheckDeltaValue := LastValue.ULINT_T - Value.ULINT_T >= UINT_TO_ULINT(DeltaVar);
		END_IF
		IF CheckDeltaValue THEN LastValue.ULINT_T := Value.ULINT_T; END_IF
	//VAR_TYPES.REAL_T:
	IBaseLibrary.TypeClass.TYPE_REAL:
		CheckDeltaValue := ABS(LastValue.REAL_T * Faktor - Value.REAL_T * Faktor) >= UINT_TO_REAL(DeltaVar)  ;
		IF CheckDeltaValue THEN LastValue.REAL_T := Value.REAL_T; END_IF
	//VAR_TYPES.LREAL_T:
	IBaseLibrary.TypeClass.TYPE_LREAL:
		//CheckDeltaValue := (ABS(LAST_VALUE.LREAL_T * RealFaktor) + UINT_TO_LREAL(DeltaVar)) <= ABS(Value.LREAL_T * RealFaktor);
		CheckDeltaValue := ABS(LastValue.LREAL_T * Faktor - Value.LREAL_T * Faktor) >= UINT_TO_LREAL(DeltaVar)  ;
		IF CheckDeltaValue THEN LastValue.LREAL_T := Value.LREAL_T; END_IF
	//VAR_TYPES.BYTE_T:
	IBaseLibrary.TypeClass.TYPE_BYTE:
		CheckDeltaValue := ABS(BYTE_TO_INT(LastValue.BYTE_T) - BYTE_TO_INT(Value.BYTE_T)) >= UINT_TO_INT(DeltaVar);
		IF CheckDeltaValue THEN LastValue.BYTE_T := Value.BYTE_T; END_IF
	//VAR_TYPES.WORD_T:
	IBaseLibrary.TypeClass.TYPE_WORD:
		CheckDeltaValue := ABS(WORD_TO_DINT(LastValue.WORD_T) - WORD_TO_DINT(Value.WORD_T)) >= DeltaVar;
		IF CheckDeltaValue THEN LastValue.WORD_T := Value.WORD_T; END_IF
	//VAR_TYPES.DWORD_T:
	IBaseLibrary.TypeClass.TYPE_DWORD:
		CheckDeltaValue := ABS(DWORD_TO_LINT(LastValue.DWORD_T) - DWORD_TO_LINT(Value.DWORD_T)) >= DeltaVar;
		IF CheckDeltaValue THEN LastValue.DWORD_T := Value.DWORD_T; END_IF
	//VAR_TYPES.LWORD_T:
	IBaseLibrary.TypeClass.TYPE_LWORD:
	//here we use no expand but check min max because no bigger data type...
		IF LastValue.LWORD_T <= Value.LWORD_T THEN
			CheckDeltaValue := Value.LWORD_T - LastValue.LWORD_T >= UINT_TO_ULINT(DeltaVar);	
		ELSE
			CheckDeltaValue := LastValue.LWORD_T - Value.LWORD_T >= UINT_TO_ULINT(DeltaVar);
		END_IF
		IF CheckDeltaValue THEN LastValue.LWORD_T := Value.LWORD_T; END_IF
	//VAR_TYPES.DATE_T:
	IBaseLibrary.TypeClass.TYPE_DATE:
		CheckDeltaValue := ABS(DATE_TO_LINT(LastValue.DATE_T) - DATE_TO_LINT(Value.DATE_T)) >= DeltaVar;
		IF CheckDeltaValue THEN LastValue.DATE_T := Value.DATE_T; END_IF
		
END_CASE

END_FUNCTION

// Common/Functions/GetValueFromPointer
FUNCTION GetValueFromPointer :  ALL_TYPES_UNION
VAR_INPUT
	PointerToValue:ALL_TYPES_UNION_POINTER;
	//TypeOfValue: VAR_TYPES;
	TypeOfValue: IBaseLibrary.TypeClass;
	
END_VAR
VAR
END_VAR

(*	SINT_T, USINT_T, INT_T, UINT_T, DINT_T, UDINT_T, 
				LINT_T, ULINT_T, REALT_T, LREAL_T*)
CASE TypeOfValue OF
	//VAR_TYPES.SINT_T:
	IBaseLibrary.TypeClass.TYPE_SINT:
		GetValueFromPointer.SINT_T := PointerToValue.POINTER_TO_SINT_T^;
	//VAR_TYPES.USINT_T:
	IBaseLibrary.TypeClass.TYPE_USINT:
		GetValueFromPointer.USINT_T := PointerToValue.POINTER_TO_USINT_T^;
	//VAR_TYPES.INT_T:
	IBaseLibrary.TypeClass.TYPE_INT:
		GetValueFromPointer.INT_T := PointerToValue.POINTER_TO_INT_T^;
	//VAR_TYPES.UINT_T:
	IBaseLibrary.TypeClass.TYPE_UINT:
		GetValueFromPointer.UINT_T := PointerToValue.POINTER_TO_UINT_T^;
	//VAR_TYPES.DINT_T:
	IBaseLibrary.TypeClass.TYPE_DINT:
		GetValueFromPointer.DINT_T := PointerToValue.POINTER_TO_DINT_T^;
	//VAR_TYPES.UDINT_T:
	IBaseLibrary.TypeClass.TYPE_UDINT:
		GetValueFromPointer.UDINT_T := PointerToValue.POINTER_TO_UDINT_T^;
	//VAR_TYPES.LINT_T:
	IBaseLibrary.TypeClass.TYPE_LINT:
		GetValueFromPointer.LINT_T := PointerToValue.POINTER_TO_LINT_T^;
	//VAR_TYPES.ULINT_T:
	IBaseLibrary.TypeClass.TYPE_ULINT:
		GetValueFromPointer.ULINT_T := PointerToValue.POINTER_TO_ULINT_T^;
	//VAR_TYPES.REAL_T:
	IBaseLibrary.TypeClass.TYPE_REAL:
		GetValueFromPointer.REAL_T := PointerToValue.POINTER_TO_REAL_T^;
	//VAR_TYPES.LREAL_T:
	IBaseLibrary.TypeClass.TYPE_LREAL:
		GetValueFromPointer.LREAL_T := PointerToValue.POINTER_TO_LREAL_T^;
	//VAR_TYPES.BYTE_T:
	IBaseLibrary.TypeClass.TYPE_BYTE:
		GetValueFromPointer.BYTE_T := PointerToValue.POINTER_TO_BYTE_T^;
	//VAR_TYPES.WORD_T:
	IBaseLibrary.TypeClass.TYPE_WORD:
		GetValueFromPointer.WORD_T := PointerToValue.POINTER_TO_WORD_T^;
	//VAR_TYPES.DWORD_T:
	IBaseLibrary.TypeClass.TYPE_DWORD:
		GetValueFromPointer.DWORD_T := PointerToValue.POINTER_TO_DWORD_T^;
	//VAR_TYPES.LWORD_T:
	IBaseLibrary.TypeClass.TYPE_LWORD:
		GetValueFromPointer.LWORD_T := PointerToValue.POINTER_TO_LWORD_T^;
	//VAR_TYPES.DT_T:
	IBaseLibrary.TypeClass.TYPE_DATEANDTIME:
		GetValueFromPointer.DT_T := PointerToValue.POINTER_TO_DT_T^;
	//VAR_TYPES.TIME_T:
	IBaseLibrary.TypeClass.TYPE_TIME:
		GetValueFromPointer.TIME_T := PointerToValue.POINTER_TO_TIME_T^;
	//VAR_TYPES.LTIME_T:
	IBaseLibrary.TypeClass.TYPE_LTIME:
		GetValueFromPointer.LTIME_T := PointerToValue.POINTER_TO_LTIME_T^;
	//VAR_TYPES.TOD_T:
	IBaseLibrary.TypeClass.TYPE_TIMEOFDAY:
		GetValueFromPointer.TOD_T := PointerToValue.POINTER_TO_TOD_T^;
	//VAR_TYPES.BOOL_T:
	IBaseLibrary.TypeClass.TYPE_BOOL:
		GetValueFromPointer.BOOL_T := PointerToValue.POINTER_TO_BOOL_T^;
	//VAR_TYPES.DATE_T:
	IBaseLibrary.TypeClass.TYPE_DATE:
		GetValueFromPointer.DATE_T := PointerToValue.POINTER_TO_DATE_T^;
	
END_CASE

END_FUNCTION

// Common/Functions/GetValueString
FUNCTION GetValueString : STRING
VAR_INPUT
	VALUE:ALL_TYPES_UNION;
	TypeOfValue:IBaseLibrary.TypeClass;
	//TypeOfValue:VAR_TYPES;
	
	DecimalPlace:INT;
END_VAR
VAR
END_VAR

(*	SINT_T, USINT_T, INT_T, UINT_T, DINT_T, UDINT_T, 
				LINT_T, ULINT_T, REALT_T, LREAL_T*)
CASE TypeOfValue OF
	//VAR_TYPES.SINT_T:
	IBaseLibrary.TypeClass.TYPE_SINT:
		GetValueString := SINT_TO_STRING(VALUE.SINT_T);
	//VAR_TYPES.USINT_T:
	IBaseLibrary.TypeClass.TYPE_USINT:
		GetValueString := USINT_TO_STRING(VALUE.USINT_T);		
	//VAR_TYPES.INT_T:
	IBaseLibrary.TypeClass.TYPE_INT:
		GetValueString := INT_TO_STRING(VALUE.INT_T);
	//VAR_TYPES.UINT_T:
	IBaseLibrary.TypeClass.TYPE_UINT:
		GetValueString := UINT_TO_STRING(VALUE.UINT_T);
	//VAR_TYPES.DINT_T:
	IBaseLibrary.TypeClass.TYPE_DINT:
		GetValueString := DINT_TO_STRING(VALUE.DINT_T);
	//VAR_TYPES.UDINT_T:
	IBaseLibrary.TypeClass.TYPE_UDINT:
		GetValueString := UDINT_TO_STRING(VALUE.UDINT_T);
	//VAR_TYPES.LINT_T:
	IBaseLibrary.TypeClass.TYPE_LINT:
		GetValueString := LINT_TO_STRING(VALUE.LINT_T);
	//VAR_TYPES.ULINT_T:
	IBaseLibrary.TypeClass.TYPE_ULINT:
		GetValueString := ULINT_TO_STRING(VALUE.ULINT_T);
	//VAR_TYPES.REAL_T:
	IBaseLibrary.TypeClass.TYPE_REAL:
		GetValueString := OSCAT_BASIC.REAL_TO_STRF(VALUE.REAL_T ,DecimalPlace,'.');
	//VAR_TYPES.LREAL_T:
	IBaseLibrary.TypeClass.TYPE_LREAL:
		GetValueString := BASIC_Extension.LREAL_TO_STRF(VALUE.LREAL_T ,DecimalPlace,'.');
	//VAR_TYPES.BYTE_T:
	IBaseLibrary.TypeClass.TYPE_BYTE:
		GetValueString := BYTE_TO_STRING(VALUE.BYTE_T);
	//VAR_TYPES.WORD_T:
	IBaseLibrary.TypeClass.TYPE_WORD:
		GetValueString := WORD_TO_STRING(VALUE.WORD_T);
	//VAR_TYPES.DWORD_T:
	IBaseLibrary.TypeClass.TYPE_DWORD:
		GetValueString := DWORD_TO_STRING(VALUE.DWORD_T);
	//VAR_TYPES.LWORD_T:
	IBaseLibrary.TypeClass.TYPE_LWORD:
		GetValueString := LWORD_TO_STRING(VALUE.LWORD_T);
	//VAR_TYPES.DT_T:
	IBaseLibrary.TypeClass.TYPE_DATEANDTIME:
		GetValueString := DT_TO_STRING(VALUE.DT_T);
	//VAR_TYPES.TIME_T:
	IBaseLibrary.TypeClass.TYPE_TIME:
		GetValueString := TIME_TO_STRING(VALUE.TIME_T);
	//VAR_TYPES.LTIME_T:
	IBaseLibrary.TypeClass.TYPE_LTIME:
		GetValueString := LTIME_TO_STRING(VALUE.LTIME_T);
	//VAR_TYPES.TOD_T:
	IBaseLibrary.TypeClass.TYPE_TIMEOFDAY:
		GetValueString := TOD_TO_STRING(VALUE.TOD_T);
	//VAR_TYPES.BOOL_T:
	IBaseLibrary.TypeClass.TYPE_BOOL:
		GetValueString := OSCAT_BASIC.LOWERCASE(str:=  BOOL_TO_STRING(VALUE.BOOL_T));
	//VAR_TYPES.DATE_T:
	IBaseLibrary.TypeClass.TYPE_DATE:
		GetValueString := DATE_TO_STRING(VALUE.DATE_T);
END_CASE

END_FUNCTION

// Common/Function Blocks/CounterToActuall
FUNCTION_BLOCK CounterToActuall
VAR_INPUT

END_VAR
VAR_OUTPUT
	//actuell consumtion
	Actuell:LREAL;
	//consumption of counter
	Counters:ARRAY[0..MyConstants.COUNTER_COUNT-1]OF LREAL;
	//consumption at reset
	CountersValueAtReset:ARRAY[0..MyConstants.COUNTER_COUNT-1]OF LREAL;
	//actuell average Value
	CountersAverageValue:ARRAY[0..MyConstants.COUNTER_COUNT-1]OF LREAL;
	//counts of impuls
	Counts:ARRAY[0..MyConstants.COUNTER_COUNT-1]OF LREAL;
END_VAR
VAR
	CounterFaktor:LREAL;
	//time base for Counter val in s
	CounterTimeBase:LREAL;
	//impulse of Counter
	Pulse:POINTER TO BOOL;
	LastImp:CAA.TICK;
	RTrig:R_TRIG;
	CounterResetPointer:ARRAY[0..MyConstants.COUNTER_COUNT-1] OF POINTER TO BOOL;
	CounterIsParam:ARRAY[0..MyConstants.COUNTER_COUNT-1] OF BOOL;
	CounterEdge:ARRAY[0..MyConstants.COUNTER_COUNT-1]OF R_TRIG;
	i:UINT;
END_VAR

RTrig(CLK:= Pulse^);
IF RTrig.Q THEN
	Actuell := (CounterFaktor * CounterTimeBase) / (TO_LREAL(Time_and_Date.TICKS.GetTick(xDummy:= TRUE) - LastImp)/1000);
	LastImp := Time_and_Date.TICKS.GetTick(xDummy:= TRUE);
	//increase counters
	FOR i:=0 TO MyConstants.COUNTER_COUNT -1 DO
		Counters[i] := Counters[i] + CounterFaktor;
		Counts[i] := Counts[i] + 1;
		CountersAverageValue[i] := Counters[i] / Counts[i];  
	END_FOR
END_IF
//check if i have to reset counters....
FOR i:=0 TO MyConstants.COUNTER_COUNT -1 DO
	IF CounterIsParam[i] THEN
		CounterEdge[i](CLK:= CounterResetPointer[i]^);
		IF CounterEdge[i].Q THEN
			CountersValueAtReset[i] := Counters[i];
			Counters[i] := 0;
			Counts[i] := 0;
		END_IF
	END_IF
END_FOR

METHOD CounterInit
VAR_INPUT
	CounterFaktor:LREAL;
	//time base for Counter val in s
	CounterTimeBase:LREAL;
	//impulse of Counter
	Pulse:POINTER TO BOOL;
END_VAR
THIS^.CounterFaktor := CounterFaktor;
	
THIS^.CounterTimeBase := CounterTimeBase;

THIS^.Pulse :=	Pulse;
END_METHOD

METHOD SetCounterResetImp
VAR_INPUT
ImpVar:POINTER TO BOOL;
CounterNum:UINT;

END_VAR
IF  CounterNum < MyConstants.COUNTER_COUNT - 1 THEN
	CounterResetPointer[CounterNum] := ImpVar;
	CounterIsParam[CounterNum] := TRUE;
END_IF
END_METHOD

END_FUNCTION_BLOCK

// Common/Functions/test
FUNCTION test : bool
VAR_INPUT
END_VAR
VAR
	un:ALL_TYPES_UNION_POINTER:=(POINTER_TO_LREAL_T:=ADR(r1));
	
	r1:LREAL;
	//ar1:ARRAY[0..5] OF ALL_TYPES_UNION_POINTER[(ADR(r1))];
	
	pw1:PWConfigs:=(PointerTo:=( POINTER_TO_LREAL_T:=ADR(r1)));
	apw1:ARRAY[0..1]OF PWConfigs:=[(PointerTo:=( POINTER_TO_LREAL_T:=ADR(r1)))];
END_VAR

END_FUNCTION

// Common/Functions/StrEquals
//returns true if strings equals, else false
FUNCTION StrEquals : bool
VAR_INPUT
	str1:POINTER TO STRING;
	str2:POINTER TO STRING;
END_VAR
VAR
	
	pt1:POINTER TO BYTE;
	pt2:POINTER TO BYTE;
END_VAR

StrEquals := TRUE;

pt1 := str1;
pt2 := str2;
WHILE pt1^ <> 0 DO 
	IF pt1^ <> pt2^ THEN
		StrEquals := FALSE;
		EXIT;
	END_IF
	pt1 := pt1 + SIZEOF(BYTE);
	pt2 := pt2 + SIZEOF(BYTE);
END_WHILE
//check if string 2 is at end to, if not, so not equal

IF pt2^ <> 0 THEN
	StrEquals := FALSE;
END_IF

END_FUNCTION

// Common/Functions/StrEqualsAtStart
//returns true if strings equals, else false
FUNCTION StrEqualsAtStart : bool
VAR_INPUT
	//needs to be the shorter string, this is the depending lenght
	str1:POINTER TO STRING;
	//scond String, is longer one with to check
	str2:POINTER TO STRING;
END_VAR
VAR
	
	pt1:POINTER TO BYTE;
	pt2:POINTER TO BYTE;
END_VAR

StrEqualsAtStart := TRUE;

pt1 := str1;
pt2 := str2;
WHILE pt1^ <> 0 DO 
	IF pt1^ <> pt2^ THEN
		StrEqualsAtStart := FALSE;
		EXIT;
	END_IF
	pt1 := pt1 + SIZEOF(BYTE);
	pt2 := pt2 + SIZEOF(BYTE);
END_WHILE

END_FUNCTION

// Common/Functions/GetValueFromStringPt
FUNCTION GetValueFromStringPt : BOOL
VAR_INPUT
	//type of var
	TypeOfValue:IBaseLibrary.TypeClass;
	//pointer to target
	Target:ALL_TYPES_UNION_POINTER;
	
	//value as string
	str:POINTER TO STRING(2000);
	
END_VAR
VAR
END_VAR

(*	SINT_T, USINT_T, INT_T, UINT_T, DINT_T, UDINT_T, 
				LINT_T, ULINT_T, REALT_T, LREAL_T*)
CASE TypeOfValue OF
	//VAR_TYPES.SINT_T:
	IBaseLibrary.TypeClass.TYPE_SINT:
		Target.POINTER_TO_SINT_T^ := STRING_TO_SINT(str^);
	//VAR_TYPES.USINT_T:
	IBaseLibrary.TypeClass.TYPE_USINT:
		Target.POINTER_TO_USINT_T^ := STRING_TO_USINT(str^);		
	//VAR_TYPES.INT_T:
	IBaseLibrary.TypeClass.TYPE_INT:
		Target.POINTER_TO_INT_T^ := STRING_TO_INT(str^);
	//VAR_TYPES.UINT_T:
	IBaseLibrary.TypeClass.TYPE_UINT:
		Target.POINTER_TO_UINT_T^ := STRING_TO_UINT(str^);
	//VAR_TYPES.DINT_T:
	IBaseLibrary.TypeClass.TYPE_DINT:
		Target.POINTER_TO_DINT_T^ := STRING_TO_DINT(str^);
	//VAR_TYPES.UDINT_T:
	IBaseLibrary.TypeClass.TYPE_UDINT:
		Target.POINTER_TO_UDINT_T^ := STRING_TO_UDINT(str^);
	//VAR_TYPES.LINT_T:
	IBaseLibrary.TypeClass.TYPE_LINT:
		AtomicWriteLInt(pDest:= Target.POINTER_TO_LINT_T, liValue:= STRING_TO_LINT(str^));
		//Target.POINTER_TO_LINT_T^ := STRING_TO_LINT(str^);
	//VAR_TYPES.ULINT_T:
	IBaseLibrary.TypeClass.TYPE_ULINT:
		AtomicWriteULInt(pDest:= Target.POINTER_TO_ULINT_T, uliValue:= STRING_TO_ULINT(str^));
		//Target.POINTER_TO_ULINT_T^ := STRING_TO_ULINT(str^);
	//VAR_TYPES.REAL_T:
	IBaseLibrary.TypeClass.TYPE_REAL:
		Target.POINTER_TO_REAL_T^ := STRING_TO_REAL(str^);
	//VAR_TYPES.LREAL_T:
	IBaseLibrary.TypeClass.TYPE_LREAL:
		AtomicWriteLReal(pDest:= Target.POINTER_TO_LREAL_T, lrValue:= STRING_TO_LREAL(str^));
		//Target.POINTER_TO_LREAL_T^ := STRING_TO_LREAL(str^);
	//VAR_TYPES.BYTE_T:
	IBaseLibrary.TypeClass.TYPE_BYTE:
		Target.POINTER_TO_BYTE_T^ := STRING_TO_BYTE(str^);
	//VAR_TYPES.WORD_T:
	IBaseLibrary.TypeClass.TYPE_WORD:
		Target.POINTER_TO_WORD_T^ := STRING_TO_WORD(str^);
	//VAR_TYPES.DWORD_T:
	IBaseLibrary.TypeClass.TYPE_DWORD:
		Target.POINTER_TO_DWORD_T^ := STRING_TO_DWORD(str^);
	//VAR_TYPES.LWORD_T:
	IBaseLibrary.TypeClass.TYPE_LWORD:
		AtomicWriteLWord(pDest:= Target.POINTER_TO_LWORD_T, lwValue:= STRING_TO_LWORD(str^));
		//Target.POINTER_TO_LWORD_T^ := STRING_TO_LWORD(str^);
	//VAR_TYPES.DT_T:
	IBaseLibrary.TypeClass.TYPE_DATEANDTIME:
		Target.POINTER_TO_DT_T^ := STRING_TO_DT(str^);
	//VAR_TYPES.TIME_T:
	IBaseLibrary.TypeClass.TYPE_TIME:
		Target.POINTER_TO_TIME_T^ := STRING_TO_TIME(str^);
	//VAR_TYPES.LTIME_T:
	IBaseLibrary.TypeClass.TYPE_LTIME:
		AtomicWriteLTime(pDest:= Target.POINTER_TO_LTIME_T, ltValue:= STRING_TO_LTIME(str^));
		//Target.POINTER_TO_TIME_T^ := STRING_TO_TIME(str^);
	//VAR_TYPES.TOD_T:
	IBaseLibrary.TypeClass.TYPE_TIMEOFDAY:
		Target.POINTER_TO_TOD_T^ := STRING_TO_TOD(str^);
	//VAR_TYPES.BOOL_T:
	IBaseLibrary.TypeClass.TYPE_BOOL:
		Target.POINTER_TO_BOOL_T^ := STRING_TO_BOOL(str^);
	//VAR_TYPES.DATE_T:
	IBaseLibrary.TypeClass.TYPE_DATE:
		Target.POINTER_TO_DATE_T^ := STRING_TO_DATE(str^);
	//VAR_TYPES.STRING_T:
	IBaseLibrary.TypeClass.TYPE_STRING:
		Target.POINTER_TO_STRING_T^ := str^;
	
END_CASE

END_FUNCTION

// Common/Functions/StrEqualsAtStartWithDelimiter
//returns true if string at start equals and next char in string 2 is delim chart, else false
FUNCTION StrEqualsAtStartWithDelimiter : bool
VAR_INPUT
	//needs to be the shorter string, this is the depending lenght
	str1:POINTER TO STRING;
	//scond String, is longer one with to check
	str2:POINTER TO STRING;
	//split char/ Delmiter
	delimiter : BYTE;
END_VAR
VAR
	
	pt1:POINTER TO BYTE;
	pt2:POINTER TO BYTE;
END_VAR

StrEqualsAtStartWithDelimiter := TRUE;

pt1 := str1;
pt2 := str2;
WHILE pt1^ <> 0 AND pt2^<> 0 DO 
	IF pt1^ <> pt2^ THEN
		StrEqualsAtStartWithDelimiter := FALSE;
		EXIT;
	END_IF
	pt1 := pt1 + SIZEOF(BYTE);
	pt2 := pt2 + SIZEOF(BYTE);
END_WHILE
IF pt2^ <> delimiter THEN
	StrEqualsAtStartWithDelimiter := FALSE;
END_IF

END_FUNCTION

// Common/Functions/FindLastDot
FUNCTION FindLastDot : POINTER TO STRING(255)
VAR_INPUT
	str:POINTER TO STRING;
END_VAR
VAR
	pt:POINTER TO BYTE;
	c:BYTE;
END_VAR

c := GetChar('.');

pt := str;

WHILE pt^ <> 0 DO
	IF pt^ = c THEN
		FindLastDot := pt;
	END_IF
	pt := pt + SIZEOF(BYTE);
END_WHILE

END_FUNCTION

// Common/Functions/MakeAllTypesPointer
//returns a ALL_TYPES_UNION_POINTER from a dedicatet union

FUNCTION MakeAllTypesPointer : ALL_TYPES_UNION_POINTER
VAR_INPUT
	myType:IBaseLibrary.TypeClass;
	//myType:VAR_TYPES;
	
	fromWho:POINTER TO ALL_TYPES_UNION;
END_VAR
VAR
END_VAR

CASE myType OF
	//VAR_TYPES.SINT_T:
	IBaseLibrary.TypeClass.TYPE_SINT:
		MakeAllTypesPointer.POINTER_TO_SINT_T := ADR(fromWho^.SINT_T);
	//VAR_TYPES.USINT_T:
	IBaseLibrary.TypeClass.TYPE_USINT:
		MakeAllTypesPointer.POINTER_TO_USINT_T := ADR(fromWho^.USINT_T);
	//VAR_TYPES.INT_T:
	IBaseLibrary.TypeClass.TYPE_INT:
		MakeAllTypesPointer.POINTER_TO_INT_T := ADR(fromWho^.INT_T);
	//VAR_TYPES.UINT_T:
	IBaseLibrary.TypeClass.TYPE_UINT:
		MakeAllTypesPointer.POINTER_TO_UINT_T := ADR(fromWho^.UINT_T);
	//VAR_TYPES.DINT_T:
	IBaseLibrary.TypeClass.TYPE_DINT:
		MakeAllTypesPointer.POINTER_TO_DINT_T := ADR(fromWho^.DINT_T);
	//VAR_TYPES.UDINT_T:
	IBaseLibrary.TypeClass.TYPE_UDINT:
		MakeAllTypesPointer.POINTER_TO_UDINT_T := ADR(fromWho^.UDINT_T);
	//VAR_TYPES.LINT_T:
	IBaseLibrary.TypeClass.TYPE_LINT:
		MakeAllTypesPointer.POINTER_TO_LINT_T := ADR(fromWho^.LINT_T);
	//VAR_TYPES.ULINT_T:
	IBaseLibrary.TypeClass.TYPE_ULINT:
		MakeAllTypesPointer.POINTER_TO_ULINT_T := ADR(fromWho^.ULINT_T);
	//VAR_TYPES.REAL_T:
	IBaseLibrary.TypeClass.TYPE_REAL:
		MakeAllTypesPointer.POINTER_TO_REAL_T := ADR(fromWho^.REAL_T);
	//VAR_TYPES.LREAL_T:
	IBaseLibrary.TypeClass.TYPE_LREAL:
		MakeAllTypesPointer.POINTER_TO_LREAL_T := ADR(fromWho^.LREAL_T);
	//VAR_TYPES.BYTE_T:
	IBaseLibrary.TypeClass.TYPE_BYTE:
		MakeAllTypesPointer.POINTER_TO_BYTE_T := ADR(fromWho^.BYTE_T);
	//VAR_TYPES.WORD_T:
	IBaseLibrary.TypeClass.TYPE_WORD:
		MakeAllTypesPointer.POINTER_TO_WORD_T := ADR(fromWho^.WORD_T);
	//VAR_TYPES.DWORD_T:
	IBaseLibrary.TypeClass.TYPE_DWORD:
		MakeAllTypesPointer.POINTER_TO_DWORD_T := ADR(fromWho^.DWORD_T);
	//VAR_TYPES.LWORD_T:
	IBaseLibrary.TypeClass.TYPE_LWORD:
		MakeAllTypesPointer.POINTER_TO_LWORD_T := ADR(fromWho^.LWORD_T);
	//VAR_TYPES.DT_T:
	IBaseLibrary.TypeClass.TYPE_DATEANDTIME:
		MakeAllTypesPointer.POINTER_TO_DT_T := ADR(fromWho^.DT_T);
	//VAR_TYPES.TIME_T:
	IBaseLibrary.TypeClass.TYPE_TIME:
		MakeAllTypesPointer.POINTER_TO_TIME_T := ADR(fromWho^.TIME_T);
	//VAR_TYPES.TOD_T:
	IBaseLibrary.TypeClass.TYPE_TIMEOFDAY:
		MakeAllTypesPointer.POINTER_TO_TOD_T := ADR(fromWho^.TOD_T);
	//VAR_TYPES.BOOL_T:
	IBaseLibrary.TypeClass.TYPE_BOOL:
		MakeAllTypesPointer.POINTER_TO_BOOL_T := ADR(fromWho^.BOOL_T);
	//VAR_TYPES.DATE_T:
	IBaseLibrary.TypeClass.TYPE_DATE:
		MakeAllTypesPointer.POINTER_TO_DATE_T := ADR(fromWho^.DATE_T);
	
END_CASE

END_FUNCTION

// Common/Function Blocks/StringImpact
FUNCTION_BLOCK StringImpact
VAR_INPUT
END_VAR
VAR_OUTPUT
END_VAR
VAR
	s1:STRING(10):='ABCDEFGHIJ';
	s2:STRING(5);
	s3:STRING(5);
	p1:POINTER TO STRING(10);
	p2:POINTER TO STRING(10);
END_VAR

p1 := ADR(s1);
p2 := ADR(s2);
p2^:= p1^;

END_FUNCTION_BLOCK

// Common/Function Blocks/GetInstanceName
{attribute 'reflection'}
FUNCTION_BLOCK GetInstanceName

//this is needed for FBinstance name in Variable
VAR_INPUT
END_VAR
VAR_OUTPUT
END_VAR
VAR
	{attribute 'instance-path'}
	{attribute 'noinit'}
	instanceName: STRING(255);//this string contains the instance name of the FB
	//here we get the "lowest" element of the name...
END_VAR

(*returns the instancename of calling instance as MQTT topic,
works only with string length < 255*)
METHOD GetInstanceTopic : string(255)
VAR_INPUT
END_VAR
VAR
	BytePt:POINTER TO BYTE;
END_VAR
GetInstanceTopic := instanceName;
//now delete last instance --> this

BytePt := FindLastDot(str:= ADR(GetInstanceTopic));
BytePt^ := 0; 

//now replace all  dots with "/"

GetInstanceTopic := OSCAT_BASIC.REPLACE_ALL(str:= GetInstanceTopic, src:= '.', rep:= '/');
//done...
END_METHOD

METHOD ReduceToLastNLevels : STRING(255)
VAR_INPUT
	Level:USINT;
END_VAR
VAR
	
	cmpByte:BYTE;
	bytePointer:POINTER TO BYTE;
	StringPointer:POINTER TO STRING;
	i:UINT;
END_VAR

cmpByte:= GetChar('.');

ReduceToLastNLevels := instanceName;

bytePointer :=  FindLastDot(str:= ADR(ReduceToLastNLevels));
bytePointer^ := 0;
//bytePointer := ADR(ReduceToLastNLevels) + len(str:= ADR(ReduceToLastNLevels));
bytePointer := bytePointer - 1;
i := 0;

WHILE bytePointer >= ADR(ReduceToLastNLevels) DO
	IF bytePointer^ = cmpByte THEN
		i := i + 1; 
	END_IF
	
	IF i = Level THEN
		
		StringPointer := bytePointer + 1;
		ReduceToLastNLevels := StringPointer^; 
		RETURN;
	END_IF
	bytePointer := bytePointer - 1;
END_WHILE
END_METHOD

METHOD getLastName : string
VAR_INPUT
END_VAR
VAR
	tmpString:STRING(255);
	
	StrPt:POINTER TO STRING;
END_VAR
tmpString := instanceName;

StrPt := FindLastDot(str:= ADR(tmpString));
StrPt := StrPt + 1; 
getLastName := StrPt^;
END_METHOD

METHOD GetName : string(255)
VAR_INPUT
END_VAR
GetName := instanceName;
END_METHOD

END_FUNCTION_BLOCK

// Common/Functions/GetJSONValue
FUNCTION GetJSONValue : string(255)
VAR_INPUT
	fromWhere:POINTER TO STRING(65000);
END_VAR
VAR
	pt1: POINTER TO BYTE;
	pt2: POINTER TO BYTE;
	compByte1: BYTE;
	compByte2: BYTE;
	compByte3: BYTE;
END_VAR

// first find :

compByte1 := GetChar(':');
compByte2 := GetChar('"');
compByte3 := GetChar('}');

WHILE pt1^ <> compByte1 DO 
	pt1 := pt1 + 1;
END_WHILE


//check if '"' is next 

pt1 := pt1 + 1;

IF pt1^ = GetChar('"') THEN
	//add a 1
	pt1 := pt1 + 1;
END_IF

//here search for ',' or '}' or '"'

pt2 := pt1;

WHILE pt2^ <> compByte1 AND pt2^ <> compByte2 AND pt2^ <> compByte3 DO 
	pt2 := pt2 + 1;
END_WHILE

//so now we can copy the string...

SysMem.SysMemCpy(pDest:= ADR(GetJSONValue), pSrc:= pt1, udiCount:= pt2 - pt1);
//now add trailing zero

pt2 := pt2 + 1;
pt2^:= 0;

END_FUNCTION

// Common/Function Blocks/RELAIS_OUT_16_TRANSLATOR
FUNCTION_BLOCK RELAIS_OUT_16_TRANSLATOR
VAR_INPUT
	outs:ARRAY[0..1] OF BYTE;
	target:POINTER TO ARRAY[0..1] OF BYTE;//I2C_MUX.PCF8575OUT;
END_VAR
VAR_OUTPUT
END_VAR
VAR
	temp0 : BYTE;
	temp1 : BYTE;
END_VAR
(*
translates data to an 16 bit relais output
output:
channel - bit
16 0.0
14 0.1
12 0.2
10 0.3
8 0.4
6 0.5
4 0.6
2 0.7
1 1.0
3 1.1
5 1.2
7 1.3
9 1.4
11 1.5
13 1.6
15 1.7

*)

temp0 := NOT outs[0];
temp1 := NOT outs[1];
target^[0].0 :=temp1.7;
target^[0].1 :=temp1.5;
target^[0].2 :=temp1.3;
target^[0].3 :=temp1.1;
target^[0].4 :=temp0.7;
target^[0].5 :=temp0.5;
target^[0].6 :=temp0.3;
target^[0].7 :=temp0.1;

target^[1].0 :=temp0.0;
target^[1].1 :=temp0.2;
target^[1].2 :=temp0.4;
target^[1].3 :=temp0.6;
target^[1].4 :=temp1.0;
target^[1].5 :=temp1.2;
target^[1].6 :=temp1.4;
target^[1].7 :=temp1.6;

END_FUNCTION_BLOCK

// Common/Function Blocks/SmartDim
FUNCTION_BLOCK SmartDim
VAR_INPUT
	start:BOOL;
	delayUntilDown:TIME;
	DataUp:POINTER TO SMART_DIMM;
	DataDown:POINTER TO SMART_DIMM;
END_VAR
VAR_OUTPUT
END_VAR
VAR
	aktStage:USINT;
	timerUntilOff:tof;
	LastTime:UINT;
	isOn: BOOL;
	StageTimer:ton;
	tmpOut:REAL;
END_VAR


IF start THEN
	IF NOT isOn THEN
		StageTimer(IN:= TRUE, PT:= DataUp^.values[aktStage].RunTime);
		tmpOut := OSCAT_BASIC.SCALE_R(
			X:= TO_REAL(StageTimer.ET), 
			I_LO:= DataUp^.values[aktStage]._from, 
			I_HI:= DataUp^.values[aktStage]._to, 
			O_LO:= DataUp^.values[aktStage]._from, 
			O_HI:= DataUp^.values[aktStage]._to);
	
	END_IF
	

END_IF

IF NOT isOn THEN
	;
END_IF

END_FUNCTION_BLOCK

// Common/Functions/Steps
FUNCTION Steps : real
VAR_INPUT
	aktVal:REAL;
	lastVal:REAL;
	stepsIn:REAL;
	base:REAL;
	mode: BOOL;//true --> up, false --> down
	
END_VAR
VAR
	aktFaktor:INT;
END_VAR

IF mode THEN
	aktFaktor := TO_INT((aktVal - base) / stepsIn);
	IF aktFaktor * StepsIn + base > aktVal THEN
		Steps := aktVal;
	ELSE
		Steps := lastVal;
	END_IF
ELSE
	;
END_IF

END_FUNCTION

// Common/Function Blocks/Spratzel
FUNCTION_BLOCK Spratzel
VAR_INPUT
	on: BOOL;
	onSpratzel:BOOL:=FALSE;
END_VAR
VAR_OUTPUT
	//otuput
	Out: BOOL;
	//spratzel is on
	isOn: BOOL;

END_VAR
VAR
	myRand:Rand;
	spratzelCount:INT;
	//aktuelle anzahl Spratzel
	aktSpratzel:INT;
	step:INT;
	start:r_trig;
	stop:f_trig;
	verz:ton;
	verzZeit:TIME;
	startTimer: BOOL;

END_VAR

start(clk:= on);
stop(clk:= on);
IF start.Q THEN
	step :=5;
	//anzahl der Spratzels ermitteln
	spratzelCount := myRand.getRand(HighIn:= 4, LowIn:= 1);
	verzZeit := INT_TO_TIME(myRand.getRand(HighIn:= 800, LowIn:= 100));
	startTimer := TRUE;
	aktSpratzel := 0;
END_IF
IF stop.Q THEN
	step := 0;
	out := FALSE;
	isOn := FALSE;
END_IF

verz(IN:= startTimer, pt:= verzZeit);
CASE step OF
	5:
	IF verz.Q THEN
		IF aktSpratzel >= spratzelCount THEN
			verz(IN:= FALSE, pt:= verzZeit);
			step := 15;
			isOn := TRUE;
			startTimer := FALSE;
		ELSE
			verz(IN:= FALSE, pt:= verzZeit);
			verzZeit := INT_TO_TIME(myRand.getRand(HighIn:= 800, LowIn:= 100));
			step := 10;
		END_IF
		out := TRUE;
	END_IF
	10:
	IF verz.Q THEN
		verz(IN:= FALSE, pt:= verzZeit);
		verzZeit := INT_TO_TIME(myRand.getRand(HighIn:= 800, LowIn:= 100));
		out := FALSE;
		step := 5;
		aktSpratzel := aktSpratzel + 1;
	END_IF
	15:
		;
END_CASE

METHOD setRand
VAR_INPUT
	newRand:Rand;
END_VAR
myRand := newRand;
END_METHOD

END_FUNCTION_BLOCK

// Common/Function Blocks/Rand
FUNCTION_BLOCK Rand
VAR_INPUT
END_VAR
VAR_OUTPUT
END_VAR
VAR
	myLast:INT;
END_VAR

METHOD getRand : INT
VAR_INPUT
	HighIn:INT;
	LowIn:int;
END_VAR
getRand := OSCAT_BASIC.RDM2(last:= MyLast, low:= HighIn, high:= LowIn);
END_METHOD

END_FUNCTION_BLOCK

// Common/Function Blocks/Tests/TestNames1
FUNCTION_BLOCK TestNames1
VAR_INPUT
END_VAR
VAR_OUTPUT
END_VAR
VAR
	name1:GetInstanceName;
END_VAR

END_FUNCTION_BLOCK

// Common/Function Blocks/Tests/TestInstanceName
FUNCTION_BLOCK TestInstanceName EXTENDS TestNames1
VAR_INPUT
END_VAR
VAR_OUTPUT
	//true if last names are correct.
	ok: BOOL;

END_VAR
VAR
	name2:GetInstanceName;
	
END_VAR

//FB_Init ist immer implizit verfügbar und wird primär für die Initialisierung verwendet.
//Der Rückgabewert wird nicht ausgewertet. Für gezielte Einflussnahme können Sie
//die Methoden explizit deklarieren und darin mit dem Standard-Initialisierungscode 
//zusätzlichen Code bereitstellen. Sie können den Rückgabewert auswerten.
METHOD FB_Init: BOOL
VAR_INPUT    
bInitRetains: BOOL; // TRUE: Die Retain-Variablen werden initialisiert (Reset warm / Reset kalt)    
bInCopyCode: BOOL;  // TRUE: Die Instanz wird danach in den Kopiercode kopiert (Online-Change)
END_VAR
OK := (name1.getLastName() = 'name1') and (name2.getLastName() = 'name2');
END_METHOD

END_FUNCTION_BLOCK

// Common/Function Blocks/Tests/TestAnyX
FUNCTION_BLOCK TestAnyX
VAR_INPUT
END_VAR
VAR_OUTPUT
END_VAR
VAR
	pt:ALL_TYPES_UNION_POINTER;
	value:ALL_TYPES_UNION;
	target:STRING;
	testOK: BOOL;
	Ergs:ARRAY[0..30]OF STRING;
END_VAR

testOK := TRUE;
pt.POINTER_TO_BOOL_T := ADR(value.BOOL_T);
value.BOOL_T := TRUE;
ergs[0] := GetValueString(VALUE:= value, TypeOfValue:= IBaseLibrary.TypeClass.TYPE_BOOL, DecimalPlace:= 0);
IF ergs[0] <> 'TRUE' THEN
	testOK := FALSE;
END_IF 
value.BYTE_T := 5;
ergs[1] := GetValueString(VALUE:= value, TypeOfValue:= IBaseLibrary.TypeClass.TYPE_BYTE, DecimalPlace:= 0);
IF ergs[1] <> '5' THEN
	testOK := FALSE;
END_IF 
value.DATE_T := D#2020-02-02;
ergs[2] := GetValueString(VALUE:= value, TypeOfValue:= IBaseLibrary.TypeClass.TYPE_DATE, DecimalPlace:= 0);
IF ergs[2] <> 'D#2020-02-02' THEN
	testOK := FALSE;
END_IF 
value.DINT_T := 378912458;
ergs[3] := GetValueString(VALUE:= value, TypeOfValue:= IBaseLibrary.TypeClass.TYPE_DINT, DecimalPlace:= 0);
IF ergs[3] <> '378912458' THEN
	testOK := FALSE;
END_IF 
value.DT_T := DT#2020-02-02-15:15:15;
ergs[5] := GetValueString(VALUE:= value, TypeOfValue:= IBaseLibrary.TypeClass.TYPE_DATEANDTIME, DecimalPlace:= 0);
IF ergs[5] <> 'DT#2020-02-02-15:15:15' THEN
	testOK := FALSE;
END_IF 
value.DWORD_T := 16#AABBCCDD;
ergs[6] := GetValueString(VALUE:= value, TypeOfValue:= IBaseLibrary.TypeClass.TYPE_DWORD, DecimalPlace:= 0);
IF ergs[6] <> '2864434397' THEN
	testOK := FALSE;
END_IF 
value.INT_T := -22222;
ergs[7] := GetValueString(VALUE:= value, TypeOfValue:= IBaseLibrary.TypeClass.TYPE_INT, DecimalPlace:= 0);
IF ergs[7] <> '-22222' THEN
	testOK := FALSE;
END_IF 
value.LINT_T := -1234551345143325;
ergs[8] := GetValueString(VALUE:= value, TypeOfValue:= IBaseLibrary.TypeClass.TYPE_LINT, DecimalPlace:= 0);
IF ergs[8] <> '-1234551345143325' THEN
	testOK := FALSE;
END_IF 
value.LREAL_T := 123412341.3;
ergs[9] := GetValueString(VALUE:= value, TypeOfValue:= IBaseLibrary.TypeClass.TYPE_LREAL, DecimalPlace:= 1);
IF ergs[9] <> '123412341.3' THEN
	testOK := FALSE;
END_IF 
value.LTIME_T := LTIME#1000D15H23M12S34MS2US44NS;
ergs[10] := GetValueString(VALUE:= value, TypeOfValue:= IBaseLibrary.TypeClass.TYPE_LTIME, DecimalPlace:= 0);
IF ergs[10] <> 'LTIME#1000d15h23m12s34ms2us44ns' THEN
	testOK := FALSE;
END_IF 
value.LWORD_T := 16#3ABBCCDDEEFF2211;
ergs[11] := GetValueString(VALUE:= value, TypeOfValue:= IBaseLibrary.TypeClass.TYPE_LWORD, DecimalPlace:= 0);
IF ergs[11] <> '4232201528414249489' THEN
	testOK := FALSE;
END_IF 
value.REAL_T := -12341.4;
ergs[12] := GetValueString(VALUE:= value, TypeOfValue:= IBaseLibrary.TypeClass.TYPE_REAL, DecimalPlace:= 1);
IF ergs[12] <> '-12341.4' THEN
	testOK := FALSE;
END_IF 
value.SINT_T := -66;
ergs[13] := GetValueString(VALUE:= value, TypeOfValue:= IBaseLibrary.TypeClass.TYPE_SINT, DecimalPlace:= 0);
IF ergs[13] <> '-66' THEN
	testOK := FALSE;
END_IF 
value.TIME_T := T#12H34M15S;
ergs[14] := GetValueString(VALUE:= value, TypeOfValue:= IBaseLibrary.TypeClass.TYPE_TIME, DecimalPlace:= 0);
IF ergs[14] <> 'T#12h34m15s' THEN
	testOK := FALSE;
END_IF 
value.TOD_T := TOD#15:36:30.123;
ergs[15] := GetValueString(VALUE:= value, TypeOfValue:= IBaseLibrary.TypeClass.TYPE_TIMEOFDAY, DecimalPlace:= 0);
IF ergs[15] <> 'TOD#15:36:30.123' THEN
	testOK := FALSE;
END_IF 
value.UDINT_T := 1565499482;
ergs[16] := GetValueString(VALUE:= value, TypeOfValue:= IBaseLibrary.TypeClass.TYPE_UDINT, DecimalPlace:= 0);
IF ergs[16] <> '1565499482' THEN
	testOK := FALSE;
END_IF 
value.UINT_T := 55555;
ergs[17] := GetValueString(VALUE:= value, TypeOfValue:= IBaseLibrary.TypeClass.TYPE_UINT, DecimalPlace:= 0);
IF ergs[17] <> '55555' THEN
	testOK := FALSE;
END_IF 
value.ULINT_T := 49846154646131654;
ergs[18] := GetValueString(VALUE:= value, TypeOfValue:= IBaseLibrary.TypeClass.TYPE_ULINT, DecimalPlace:= 0);
IF ergs[18] <> '49846154646131654' THEN
	testOK := FALSE;
END_IF 
value.USINT_T := 233;
ergs[19] := GetValueString(VALUE:= value, TypeOfValue:= IBaseLibrary.TypeClass.TYPE_USINT, DecimalPlace:= 0);
IF ergs[19] <> '233' THEN
	testOK := FALSE;
END_IF 
value.WORD_T := 16#ABCD;
ergs[20] := GetValueString(VALUE:= value, TypeOfValue:= IBaseLibrary.TypeClass.TYPE_WORD, DecimalPlace:= 0);
IF ergs[20] <> '43981' THEN
	testOK := FALSE;
END_IF

END_FUNCTION_BLOCK

// Common/Functions/GetValueStringFaktor
FUNCTION GetValueStringFaktor : STRING
VAR_INPUT
	VALUE:ALL_TYPES_UNION;
	TypeOfValue:IBaseLibrary.TypeClass;
	//faktor for Real Values;
	RealFaktor:INT;
	DecimalPlace:INT;
END_VAR
VAR
END_VAR

